LIN {X 0,Y 474.954,Z 430.095,A -85,B 0,C 180,E1 -7279.666,E2 -7279.666} C_VEL
LIN {X 0,Y 474.759,Z 438.387,A -85,B 0,C 180,E1 -7280.308,E2 -7280.308} C_VEL
LIN {X 0,Y 474.498,Z 446.259,A -85,B 0,C 180,E1 -7281.055,E2 -7281.055} C_VEL
LIN {X 0,Y 474.238,Z 453.634,A -85,B 0,C 180,E1 -7281.908,E2 -7281.908} C_VEL
LIN {X 0,Y 474.053,Z 461.103,A -85,B 0,C 180,E1 -7282.976,E2 -7282.976} C_VEL
LIN {X 0,Y 473.911,Z 466.922,A -85,B 0,C 180,E1 -7284.043,E2 -7284.043} C_VEL
LIN {X 0,Y 473.866,Z 470.746,A -85,B 0,C 180,E1 -7284.896,E2 -7284.896} C_VEL
LIN {X 0,Y 473.815,Z 475.078,A -85,B 0,C 180,E1 -7286.174,E2 -7286.174} C_VEL
LIN {X 0,Y 473.748,Z 478.099,A -85,B 0,C 180,E1 -7287.451,E2 -7287.451} C_VEL
LIN {X 0,Y 473.726,Z 479.418,A -85,B 0,C 180,E1 -7288.301,E2 -7288.301} C_VEL
LIN {X 0,Y 473.69,Z 480.236,A -85,B 0,C 180,E1 -7289.151,E2 -7289.151} C_VEL
LIN {X 0,Y 473.674,Z 480.528,A -85,B 0,C 180,E1 -7290.001,E2 -7290.001} C_VEL
LIN {X 0,Y 473.69,Z 480.211,A -85,B 0,C 180,E1 -7290.852,E2 -7290.852} C_VEL
LIN {X 0,Y 473.726,Z 479.389,A -85,B 0,C 180,E1 -7291.702,E2 -7291.702} C_VEL
LIN {X 0,Y 473.748,Z 478.065,A -85,B 0,C 180,E1 -7292.552,E2 -7292.552} C_VEL
LIN {X 0,Y 473.799,Z 475.012,A -85,B 0,C 180,E1 -7293.829,E2 -7293.829} C_VEL
LIN {X 0,Y 473.792,Z 472.221,A -85,B 0,C 180,E1 -7294.681,E2 -7294.681} C_VEL
LIN {X 0,Y 473.911,Z 468.787,A -85,B 0,C 180,E1 -7295.533,E2 -7295.533} C_VEL
LIN {X 0,Y 473.95,Z 463.866,A -85,B 0,C 180,E1 -7296.52,E2 -7296.52} C_VEL
LIN {X 0,Y 474.145,Z 458.151,A -85,B 0,C 180,E1 -7297.453,E2 -7297.453} C_VEL
LIN {X 0,Y 474.275,Z 451.812,A -85,B 0,C 180,E1 -7298.308,E2 -7298.308} C_VEL
LIN {X 0,Y 474.514,Z 444.11,A -85,B 0,C 180,E1 -7299.163,E2 -7299.163} C_VEL
LIN {X 0,Y 474.846,Z 434.562,A -85,B 0,C 180,E1 -7300.016,E2 -7300.016} C_VEL
LIN {X 0,Y 475.091,Z 425.305,A -85,B 0,C 180,E1 -7300.657,E2 -7300.657} C_VEL
LIN {X 0,Y 475.426,Z 415.239,A -85,B 0,C 180,E1 -7301.189,E2 -7301.189} C_VEL
LIN {X 0,Y 475.61,Z 405.755,A -85,B 0,C 180,E1 -7301.562,E2 -7301.562} C_VEL
LIN {X 0,Y 475.842,Z 395.844,A -85,B 0,C 180,E1 -7301.827,E2 -7301.827} C_VEL
LIN {X 0,Y 476.275,Z 333.715,A -85,B 0,C 180,E1 -7302.911,E2 -7302.911} C_VEL
LIN {X 0,Y 474.456,Z 318.892,A -85,B 0,C 180,E1 -7303.244,E2 -7303.244} C_VEL
LIN {X 0,Y 474.728,Z 301.496,A -85,B 0,C 180,E1 -7306.338,E2 -7306.338} C_VEL
LIN {X 0,Y 475.004,Z 283.808,A -85,B 0,C 180,E1 -7309.446,E2 -7309.446} C_VEL
LIN {X 0,Y 475.142,Z 269.646,A -85,B 0,C 180,E1 -7311.932,E2 -7311.932} C_VEL
LIN {X 0,Y 474.695,Z 266.173,A -85,B 0,C 180,E1 -7312.584,E2 -7312.584} C_VEL
LIN {X 0,Y 474.603,Z 266.18,A -85,B 0,C 180,E1 -7315.433,E2 -7315.433} C_VEL
LIN {X 0,Y 474.599,Z 266.182,A -85,B 0,C 180,E1 -7318.287,E2 -7318.287} C_VEL
LIN {X 0,Y 474.581,Z 266.183,A -85,B 0,C 180,E1 -7321.22,E2 -7321.22} C_VEL
LIN {X 0,Y 474.56,Z 266.183,A -85,B 0,C 180,E1 -7324.248,E2 -7324.248} C_VEL
LIN {X 0,Y 474.541,Z 266.185,A -85,B 0,C 180,E1 -7327.39,E2 -7327.39} C_VEL
LIN {X 0,Y 474.591,Z 266.176,A -85,B 0,C 180,E1 -7329.639,E2 -7329.639} C_VEL
LIN {X 0,Y 474.579,Z 266.185,A -85,B 0,C 180,E1 -7332.939,E2 -7332.939} C_VEL
LIN {X 0,Y 474.581,Z 266.177,A -85,B 0,C 180,E1 -7335.889,E2 -7335.889} C_VEL
LIN {X 0,Y 474.614,Z 266.179,A -85,B 0,C 180,E1 -7339.044,E2 -7339.044} C_VEL
LIN {X 0,Y 474.609,Z 266.173,A -85,B 0,C 180,E1 -7341.706,E2 -7341.706} C_VEL
LIN {X 0,Y 474.632,Z 266.174,A -85,B 0,C 180,E1 -7344.723,E2 -7344.723} C_VEL
LIN {X 0,Y 474.642,Z 266.172,A -85,B 0,C 180,E1 -7347.785,E2 -7347.785} C_VEL
LIN {X 0,Y 474.616,Z 266.179,A -85,B 0,C 180,E1 -7350.888,E2 -7350.888} C_VEL
LIN {X 0,Y 474.618,Z 266.179,A -85,B 0,C 180,E1 -7353.623,E2 -7353.623} C_VEL
LIN {X 0,Y 474.649,Z 266.175,A -85,B 0,C 180,E1 -7356.64,E2 -7356.64} C_VEL
LIN {X 0,Y 474.668,Z 266.169,A -85,B 0,C 180,E1 -7360.087,E2 -7360.087} C_VEL
LIN {X 0,Y 474.765,Z 266.163,A -85,B 0,C 180,E1 -7363.661,E2 -7363.661} C_VEL
LIN {X 0,Y 474.843,Z 266.317,A -85,B 0,C 180,E1 -7364.133,E2 -7364.133} C_VEL
LIN {X 0,Y 474.62,Z 284.701,A -85,B 0,C 180,E1 -7366.779,E2 -7366.779} C_VEL
LIN {X 0,Y 476.599,Z 298.432,A -85,B 0,C 180,E1 -7367.103,E2 -7367.103} C_VEL
LIN {X 0,Y 475.902,Z 364.749,A -85,B 0,C 180,E1 -7368.281,E2 -7368.281} C_VEL
LIN {X 0,Y 475.7,Z 376.754,A -85,B 0,C 180,E1 -7368.653,E2 -7368.653} C_VEL
LIN {X 0,Y 475.451,Z 386.848,A -85,B 0,C 180,E1 -7369.133,E2 -7369.133} C_VEL
LIN {X 0,Y 475.243,Z 395.471,A -85,B 0,C 180,E1 -7369.667,E2 -7369.667} C_VEL
LIN {X 0,Y 475.08,Z 403.741,A -85,B 0,C 180,E1 -7370.309,E2 -7370.309} C_VEL
LIN {X 0,Y 474.834,Z 411.591,A -85,B 0,C 180,E1 -7371.056,E2 -7371.056} C_VEL
LIN {X 0,Y 474.563,Z 418.93,A -85,B 0,C 180,E1 -7371.908,E2 -7371.908} C_VEL
LIN {X 0,Y 474.314,Z 427.087,A -85,B 0,C 180,E1 -7373.102,E2 -7373.102} C_VEL
LIN {X 0,Y 474.192,Z 432.129,A -85,B 0,C 180,E1 -7374.041,E2 -7374.041} C_VEL
LIN {X 0,Y 473.929,Z 435.928,A -85,B 0,C 180,E1 -7374.891,E2 -7374.891} C_VEL
LIN {X 0,Y 474.022,Z 438.984,A -85,B 0,C 180,E1 -7375.745,E2 -7375.745} C_VEL
LIN {X 0,Y 473.909,Z 441.375,A -85,B 0,C 180,E1 -7376.595,E2 -7376.595} C_VEL
LIN {X 0,Y 473.83,Z 443.205,A -85,B 0,C 180,E1 -7377.446,E2 -7377.446} C_VEL
LIN {X 0,Y 473.763,Z 444.517,A -85,B 0,C 180,E1 -7378.296,E2 -7378.296} C_VEL
LIN {X 0,Y 473.693,Z 445.334,A -85,B 0,C 180,E1 -7379.146,E2 -7379.146} C_VEL
LIN {X 0,Y 473.676,Z 445.624,A -85,B 0,C 180,E1 -7379.996,E2 -7379.996} C_VEL
LIN {X 0,Y 473.693,Z 445.313,A -85,B 0,C 180,E1 -7380.846,E2 -7380.846} C_VEL
LIN {X 0,Y 473.76,Z 444.504,A -85,B 0,C 180,E1 -7381.696,E2 -7381.696} C_VEL
LIN {X 0,Y 473.804,Z 443.201,A -85,B 0,C 180,E1 -7382.546,E2 -7382.546} C_VEL
LIN {X 0,Y 473.934,Z 440.192,A -85,B 0,C 180,E1 -7383.822,E2 -7383.822} C_VEL
LIN {X 0,Y 473.923,Z 437.448,A -85,B 0,C 180,E1 -7384.674,E2 -7384.674} C_VEL
LIN {X 0,Y 474.009,Z 434.063,A -85,B 0,C 180,E1 -7385.526,E2 -7385.526} C_VEL
LIN {X 0,Y 474.304,Z 429.112,A -85,B 0,C 180,E1 -7386.525,E2 -7386.525} C_VEL
LIN {X 0,Y 474.322,Z 423.544,A -85,B 0,C 180,E1 -7387.444,E2 -7387.444} C_VEL
LIN {X 0,Y 474.513,Z 417.257,A -85,B 0,C 180,E1 -7388.298,E2 -7388.298} C_VEL
LIN {X 0,Y 474.764,Z 410.645,A -85,B 0,C 180,E1 -7389.044,E2 -7389.044} C_VEL
LIN {X 0,Y 475.018,Z 402.647,A -85,B 0,C 180,E1 -7389.791,E2 -7389.791} C_VEL
LIN {X 0,Y 475.318,Z 392.671,A -85,B 0,C 180,E1 -7390.538,E2 -7390.538} C_VEL
LIN {X 0,Y 475.531,Z 382.089,A -85,B 0,C 180,E1 -7391.126,E2 -7391.126} C_VEL
LIN {X 0,Y 475.702,Z 372.217,A -85,B 0,C 180,E1 -7391.527,E2 -7391.527} C_VEL
LIN {X 0,Y 475.842,Z 362.639,A -85,B 0,C 180,E1 -7391.793,E2 -7391.793} C_VEL
LIN {X 0,Y 476.251,Z 297.517,A -85,B 0,C 180,E1 -7392.905,E2 -7392.905} C_VEL
LIN {X 0,Y 474.524,Z 286.851,A -85,B 0,C 180,E1 -7393.15,E2 -7393.15} C_VEL
LIN {X 0,Y 474.786,Z 274.007,A -85,B 0,C 180,E1 -7396.329,E2 -7396.329} C_VEL
LIN {X 0,Y 474.746,Z 266.283,A -85,B 0,C 180,E1 -7398.3,E2 -7398.3} C_VEL
LIN {X 0,Y 474.623,Z 266.177,A -85,B 0,C 180,E1 -7401.111,E2 -7401.111} C_VEL
LIN {X 0,Y 474.61,Z 266.177,A -85,B 0,C 180,E1 -7404.489,E2 -7404.489} C_VEL
LIN {X 0,Y 474.582,Z 266.182,A -85,B 0,C 180,E1 -7407.321,E2 -7407.321} C_VEL
LIN {X 0,Y 474.574,Z 266.18,A -85,B 0,C 180,E1 -7410.226,E2 -7410.226} C_VEL
LIN {X 0,Y 474.611,Z 266.179,A -85,B 0,C 180,E1 -7413.215,E2 -7413.215} C_VEL
LIN {X 0,Y 474.557,Z 266.182,A -85,B 0,C 180,E1 -7416.319,E2 -7416.319} C_VEL
LIN {X 0,Y 474.595,Z 266.181,A -85,B 0,C 180,E1 -7419.543,E2 -7419.543} C_VEL
LIN {X 0,Y 474.568,Z 266.182,A -85,B 0,C 180,E1 -7422.228,E2 -7422.228} C_VEL
LIN {X 0,Y 474.582,Z 266.183,A -85,B 0,C 180,E1 -7425.293,E2 -7425.293} C_VEL
LIN {X 0,Y 474.584,Z 266.182,A -85,B 0,C 180,E1 -7428.209,E2 -7428.209} C_VEL
LIN {X 0,Y 474.571,Z 266.185,A -85,B 0,C 180,E1 -7431.538,E2 -7431.538} C_VEL
LIN {X 0,Y 474.586,Z 266.179,A -85,B 0,C 180,E1 -7434.721,E2 -7434.721} C_VEL
LIN {X 0,Y 474.591,Z 266.182,A -85,B 0,C 180,E1 -7437.783,E2 -7437.783} C_VEL
LIN {X 0,Y 474.553,Z 266.183,A -85,B 0,C 180,E1 -7438.959,E2 -7438.959} C_VEL
LIN {X 0,Y 473.909,Z 266.266,A -85,B 0,C 180,E1 -7439.668,E2 -7439.668} C_VEL
LIN {X 0,Y 471.103,Z 266.616,A -85,B 0,C 180,E1 -7440.819,E2 -7440.819} C_VEL
LIN {X 0,Y 468.712,Z 266.915,A -85,B 0,C 180,E1 -7441.747,E2 -7441.747} C_VEL
LIN {X 0,Y 467.671,Z 267.043,A -85,B 0,C 180,E1 -7442.463,E2 -7442.463} C_VEL
LIN {X 0,Y 467.58,Z 267.053,A -85,B 0,C 180,E1 -7442.706,E2 -7442.706} C_VEL
LIN {X 0,Y 467.554,Z 267.055,A -85,B 0,C 180,E1 -7445.109,E2 -7445.109} C_VEL
LIN {X 0,Y 467.482,Z 267.067,A -85,B 0,C 180,E1 -7447.922,E2 -7447.922} C_VEL
LIN {X 0,Y 467.569,Z 267.056,A -85,B 0,C 180,E1 -7450.689,E2 -7450.689} C_VEL
LIN {X 0,Y 467.594,Z 267.054,A -85,B 0,C 180,E1 -7454.112,E2 -7454.112} C_VEL
LIN {X 0,Y 467.641,Z 267.045,A -85,B 0,C 180,E1 -7457.853,E2 -7457.853} C_VEL
LIN {X 0,Y 467.626,Z 267.047,A -85,B 0,C 180,E1 -7461.355,E2 -7461.355} C_VEL
LIN {X 0,Y 467.694,Z 267.038,A -85,B 0,C 180,E1 -7463.961,E2 -7463.961} C_VEL
LIN {X 0,Y 467.808,Z 267.025,A -85,B 0,C 180,E1 -7467.415,E2 -7467.415} C_VEL
LIN {X 0,Y 467.82,Z 267.022,A -85,B 0,C 180,E1 -7469.999,E2 -7469.999} C_VEL
LIN {X 0,Y 467.807,Z 267.027,A -85,B 0,C 180,E1 -7472.582,E2 -7472.582} C_VEL
LIN {X 0,Y 467.692,Z 267.038,A -85,B 0,C 180,E1 -7476.036,E2 -7476.036} C_VEL
LIN {X 0,Y 467.628,Z 267.048,A -85,B 0,C 180,E1 -7478.642,E2 -7478.642} C_VEL
LIN {X 0,Y 467.637,Z 267.044,A -85,B 0,C 180,E1 -7482.144,E2 -7482.144} C_VEL
LIN {X 0,Y 467.587,Z 267.052,A -85,B 0,C 180,E1 -7485.885,E2 -7485.885} C_VEL
LIN {X 0,Y 467.563,Z 267.057,A -85,B 0,C 180,E1 -7489.309,E2 -7489.309} C_VEL
LIN {X 0,Y 467.479,Z 267.066,A -85,B 0,C 180,E1 -7492.075,E2 -7492.075} C_VEL
LIN {X 0,Y 467.554,Z 267.056,A -85,B 0,C 180,E1 -7494.888,E2 -7494.888} C_VEL
LIN {X 0,Y 467.57,Z 267.055,A -85,B 0,C 180,E1 -7497.77,E2 -7497.77} C_VEL
LIN {X 0,Y 467.515,Z 267.061,A -85,B 0,C 180,E1 -7501.048,E2 -7501.048} C_VEL
LIN {X 0,Y 467.534,Z 267.06,A -85,B 0,C 180,E1 -7504.245,E2 -7504.245} C_VEL
LIN {X 0,Y 467.497,Z 267.063,A -85,B 0,C 180,E1 -7507.19,E2 -7507.19} C_VEL
LIN {X 0,Y 467.55,Z 267.058,A -85,B 0,C 180,E1 -7510.265,E2 -7510.265} C_VEL
LIN {X 0,Y 467.568,Z 267.055,A -85,B 0,C 180,E1 -7512.574,E2 -7512.574} C_VEL
LIN {X 0,Y 467.525,Z 267.061,A -85,B 0,C 180,E1 -7516.18,E2 -7516.18} C_VEL
LIN {X 0,Y 467.542,Z 267.058,A -85,B 0,C 180,E1 -7518.725,E2 -7518.725} C_VEL
LIN {X 0,Y 467.528,Z 267.058,A -85,B 0,C 180,E1 -7521.411,E2 -7521.411} C_VEL
LIN {X 0,Y 467.52,Z 267.062,A -85,B 0,C 180,E1 -7524.264,E2 -7524.264} C_VEL
LIN {X 0,Y 467.541,Z 267.056,A -85,B 0,C 180,E1 -7527.325,E2 -7527.325} C_VEL
LIN {X 0,Y 467.529,Z 267.06,A -85,B 0,C 180,E1 -7530.672,E2 -7530.672} C_VEL
LIN {X 0,Y 467.55,Z 267.057,A -85,B 0,C 180,E1 -7533.202,E2 -7533.202} C_VEL
LIN {X 0,Y 467.555,Z 267.059,A -85,B 0,C 180,E1 -7536.474,E2 -7536.474} C_VEL
LIN {X 0,Y 467.589,Z 267.05,A -85,B 0,C 180,E1 -7539.781,E2 -7539.781} C_VEL
LIN {X 0,Y 467.566,Z 267.057,A -85,B 0,C 180,E1 -7542.511,E2 -7542.511} C_VEL
LIN {X 0,Y 467.575,Z 267.055,A -85,B 0,C 180,E1 -7545.201,E2 -7545.201} C_VEL
LIN {X 0,Y 467.629,Z 267.045,A -85,B 0,C 180,E1 -7547.859,E2 -7547.859} C_VEL
LIN {X 0,Y 467.644,Z 267.046,A -85,B 0,C 180,E1 -7551.361,E2 -7551.361} C_VEL
LIN {X 0,Y 467.704,Z 267.036,A -85,B 0,C 180,E1 -7553.967,E2 -7553.967} C_VEL
LIN {X 0,Y 467.801,Z 267.027,A -85,B 0,C 180,E1 -7557.421,E2 -7557.421} C_VEL
LIN {X 0,Y 467.831,Z 267.021,A -85,B 0,C 180,E1 -7560.004,E2 -7560.004} C_VEL
LIN {X 0,Y 467.831,Z 267.02,A -85,B 0,C 180,E1 -7562.587,E2 -7562.587} C_VEL
LIN {X 0,Y 467.696,Z 267.039,A -85,B 0,C 180,E1 -7566.042,E2 -7566.042} C_VEL
LIN {X 0,Y 467.653,Z 267.042,A -85,B 0,C 180,E1 -7568.647,E2 -7568.647} C_VEL
LIN {X 0,Y 467.644,Z 267.046,A -85,B 0,C 180,E1 -7572.149,E2 -7572.149} C_VEL
LIN {X 0,Y 467.602,Z 267.052,A -85,B 0,C 180,E1 -7575.7,E2 -7575.7} C_VEL
LIN {X 0,Y 467.61,Z 267.05,A -85,B 0,C 180,E1 -7579.312,E2 -7579.312} C_VEL
LIN {X 0,Y 467.523,Z 267.061,A -85,B 0,C 180,E1 -7582.078,E2 -7582.078} C_VEL
LIN {X 0,Y 467.552,Z 267.055,A -85,B 0,C 180,E1 -7584.893,E2 -7584.893} C_VEL
LIN {X 0,Y 467.573,Z 267.057,A -85,B 0,C 180,E1 -7587.775,E2 -7587.775} C_VEL
LIN {X 0,Y 467.562,Z 267.054,A -85,B 0,C 180,E1 -7591.048,E2 -7591.048} C_VEL
LIN {X 0,Y 467.571,Z 267.056,A -85,B 0,C 180,E1 -7594.243,E2 -7594.243} C_VEL
LIN {X 0,Y 467.518,Z 267.059,A -85,B 0,C 180,E1 -7597.185,E2 -7597.185} C_VEL
LIN {X 0,Y 467.553,Z 267.059,A -85,B 0,C 180,E1 -7600.27,E2 -7600.27} C_VEL
LIN {X 0,Y 467.544,Z 267.056,A -85,B 0,C 180,E1 -7603.749,E2 -7603.749} C_VEL
LIN {X 0,Y 467.531,Z 267.062,A -85,B 0,C 180,E1 -7606.256,E2 -7606.256} C_VEL
LIN {X 0,Y 467.556,Z 267.054,A -85,B 0,C 180,E1 -7609.736,E2 -7609.736} C_VEL
LIN {X 0,Y 467.537,Z 267.06,A -85,B 0,C 180,E1 -7612.818,E2 -7612.818} C_VEL
LIN {X 0,Y 467.576,Z 267.052,A -85,B 0,C 180,E1 -7615.763,E2 -7615.763} C_VEL
LIN {X 0,Y 467.543,Z 267.059,A -85,B 0,C 180,E1 -7618.963,E2 -7618.963} C_VEL
LIN {X 0,Y 467.545,Z 267.056,A -85,B 0,C 180,E1 -7622.228,E2 -7622.228} C_VEL
LIN {X 0,Y 467.59,Z 267.057,A -85,B 0,C 180,E1 -7625.588,E2 -7625.588} C_VEL
LIN {X 0,Y 467.624,Z 267.185,A -85,B 0,C 180,E1 -7625.885,E2 -7625.885} C_VEL
LIN {X 0,Y 468.989,Z 275.944,A -85,B 0,C 180,E1 -7627.768,E2 -7627.768} C_VEL
LIN {X 0,Y 468.477,Z 290.486,A -85,B 0,C 180,E1 -7630.731,E2 -7630.731} C_VEL
LIN {X 0,Y 467.831,Z 306.981,A -85,B 0,C 180,E1 -7634.042,E2 -7634.042} C_VEL
LIN {X 0,Y 467.465,Z 320.443,A -85,B 0,C 180,E1 -7636.695,E2 -7636.695} C_VEL
LIN {X 0,Y 469.327,Z 337.479,A -85,B 0,C 180,E1 -7637.043,E2 -7637.043} C_VEL
LIN {X 0,Y 468.775,Z 398.013,A -85,B 0,C 180,E1 -7638.105,E2 -7638.105} C_VEL
LIN {X 0,Y 468.531,Z 408.917,A -85,B 0,C 180,E1 -7638.428,E2 -7638.428} C_VEL
LIN {X 0,Y 468.221,Z 420.685,A -85,B 0,C 180,E1 -7638.968,E2 -7638.968} C_VEL
LIN {X 0,Y 467.929,Z 429.416,A -85,B 0,C 180,E1 -7639.509,E2 -7639.509} C_VEL
LIN {X 0,Y 467.709,Z 437.792,A -85,B 0,C 180,E1 -7640.16,E2 -7640.16} C_VEL
LIN {X 0,Y 467.41,Z 445.729,A -85,B 0,C 180,E1 -7640.918,E2 -7640.918} C_VEL
LIN {X 0,Y 467.18,Z 453.162,A -85,B 0,C 180,E1 -7641.785,E2 -7641.785} C_VEL
LIN {X 0,Y 466.996,Z 460.696,A -85,B 0,C 180,E1 -7642.869,E2 -7642.869} C_VEL
LIN {X 0,Y 466.822,Z 466.563,A -85,B 0,C 180,E1 -7643.952,E2 -7643.952} C_VEL
LIN {X 0,Y 466.799,Z 470.41,A -85,B 0,C 180,E1 -7644.819,E2 -7644.819} C_VEL
LIN {X 0,Y 466.706,Z 474.77,A -85,B 0,C 180,E1 -7646.116,E2 -7646.116} C_VEL
LIN {X 0,Y 466.669,Z 477.808,A -85,B 0,C 180,E1 -7647.412,E2 -7647.412} C_VEL
LIN {X 0,Y 466.634,Z 479.14,A -85,B 0,C 180,E1 -7648.275,E2 -7648.275} C_VEL
LIN {X 0,Y 466.621,Z 479.97,A -85,B 0,C 180,E1 -7649.138,E2 -7649.138} C_VEL
LIN {X 0,Y 466.603,Z 480.263,A -85,B 0,C 180,E1 -7650.001,E2 -7650.001} C_VEL
LIN {X 0,Y 466.621,Z 479.951,A -85,B 0,C 180,E1 -7650.864,E2 -7650.864} C_VEL
LIN {X 0,Y 466.634,Z 479.134,A -85,B 0,C 180,E1 -7651.728,E2 -7651.728} C_VEL
LIN {X 0,Y 466.67,Z 477.814,A -85,B 0,C 180,E1 -7652.591,E2 -7652.591} C_VEL
LIN {X 0,Y 466.692,Z 474.769,A -85,B 0,C 180,E1 -7653.887,E2 -7653.887} C_VEL
LIN {X 0,Y 466.72,Z 471.986,A -85,B 0,C 180,E1 -7654.752,E2 -7654.752} C_VEL
LIN {X 0,Y 466.828,Z 468.557,A -85,B 0,C 180,E1 -7655.617,E2 -7655.617} C_VEL
LIN {X 0,Y 466.918,Z 463.079,A -85,B 0,C 180,E1 -7656.719,E2 -7656.719} C_VEL
LIN {X 0,Y 467.092,Z 456.451,A -85,B 0,C 180,E1 -7657.784,E2 -7657.784} C_VEL
LIN {X 0,Y 467.392,Z 448.009,A -85,B 0,C 180,E1 -7658.867,E2 -7658.867} C_VEL
LIN {X 0,Y 467.731,Z 439.338,A -85,B 0,C 180,E1 -7659.733,E2 -7659.733} C_VEL
LIN {X 0,Y 467.913,Z 431.356,A -85,B 0,C 180,E1 -7660.385,E2 -7660.385} C_VEL
LIN {X 0,Y 468.171,Z 423.182,A -85,B 0,C 180,E1 -7660.926,E2 -7660.926} C_VEL
LIN {X 0,Y 468.476,Z 413.81,A -85,B 0,C 180,E1 -7661.412,E2 -7661.412} C_VEL
LIN {X 0,Y 468.683,Z 404.762,A -85,B 0,C 180,E1 -7661.763,E2 -7661.763} C_VEL
LIN {X 0,Y 468.943,Z 394.573,A -85,B 0,C 180,E1 -7662.031,E2 -7662.031} C_VEL
LIN {X 0,Y 469.412,Z 334.466,A -85,B 0,C 180,E1 -7663.116,E2 -7663.116} C_VEL
LIN {X 0,Y 467.446,Z 318.359,A -85,B 0,C 180,E1 -7663.505,E2 -7663.505} C_VEL
LIN {X 0,Y 467.802,Z 298.693,A -85,B 0,C 180,E1 -7667.036,E2 -7667.036} C_VEL
LIN {X 0,Y 468.103,Z 279.668,A -85,B 0,C 180,E1 -7670.432,E2 -7670.432} C_VEL
LIN {X 0,Y 468.156,Z 270.594,A -85,B 0,C 180,E1 -7672.044,E2 -7672.044} C_VEL
LIN {X 0,Y 467.634,Z 267.052,A -85,B 0,C 180,E1 -7672.71,E2 -7672.71} C_VEL
LIN {X 0,Y 467.544,Z 267.058,A -85,B 0,C 180,E1 -7675.845,E2 -7675.845} C_VEL
LIN {X 0,Y 467.535,Z 267.065,A -85,B 0,C 180,E1 -7678.754,E2 -7678.754} C_VEL
LIN {X 0,Y 467.548,Z 267.055,A -85,B 0,C 180,E1 -7681.744,E2 -7681.744} C_VEL
LIN {X 0,Y 467.5,Z 267.066,A -85,B 0,C 180,E1 -7684.839,E2 -7684.839} C_VEL
LIN {X 0,Y 467.546,Z 267.054,A -85,B 0,C 180,E1 -7688.048,E2 -7688.048} C_VEL
LIN {X 0,Y 467.563,Z 267.054,A -85,B 0,C 180,E1 -7691.406,E2 -7691.406} C_VEL
LIN {X 0,Y 467.56,Z 267.058,A -85,B 0,C 180,E1 -7695.049,E2 -7695.049} C_VEL
LIN {X 0,Y 467.575,Z 267.053,A -85,B 0,C 180,E1 -7698.725,E2 -7698.725} C_VEL
LIN {X 0,Y 467.566,Z 267.049,A -85,B 0,C 180,E1 -7701.953,E2 -7701.953} C_VEL
LIN {X 0,Y 467.57,Z 267.056,A -85,B 0,C 180,E1 -7705.165,E2 -7705.165} C_VEL
LIN {X 0,Y 467.593,Z 267.05,A -85,B 0,C 180,E1 -7708.258,E2 -7708.258} C_VEL
LIN {X 0,Y 467.564,Z 267.06,A -85,B 0,C 180,E1 -7711.246,E2 -7711.246} C_VEL
LIN {X 0,Y 467.607,Z 267.051,A -85,B 0,C 180,E1 -7714.395,E2 -7714.395} C_VEL
LIN {X 0,Y 467.591,Z 267.058,A -85,B 0,C 180,E1 -7716.993,E2 -7716.993} C_VEL
LIN {X 0,Y 467.637,Z 267.047,A -85,B 0,C 180,E1 -7719.774,E2 -7719.774} C_VEL
LIN {X 0,Y 467.663,Z 267.045,A -85,B 0,C 180,E1 -7722.505,E2 -7722.505} C_VEL
LIN {X 0,Y 467.769,Z 267.09,A -85,B 0,C 180,E1 -7723.961,E2 -7723.961} C_VEL
LIN {X 0,Y 467.867,Z 271.123,A -85,B 0,C 180,E1 -7724.533,E2 -7724.533} C_VEL
LIN {X 0,Y 467.683,Z 284.995,A -85,B 0,C 180,E1 -7726.543,E2 -7726.543} C_VEL
LIN {X 0,Y 469.763,Z 299.131,A -85,B 0,C 180,E1 -7726.883,E2 -7726.883} C_VEL
LIN {X 0,Y 468.979,Z 365.544,A -85,B 0,C 180,E1 -7728.105,E2 -7728.105} C_VEL
LIN {X 0,Y 468.759,Z 377.239,A -85,B 0,C 180,E1 -7728.483,E2 -7728.483} C_VEL
LIN {X 0,Y 468.501,Z 387.235,A -85,B 0,C 180,E1 -7728.97,E2 -7728.97} C_VEL
LIN {X 0,Y 468.277,Z 395.806,A -85,B 0,C 180,E1 -7729.511,E2 -7729.511} C_VEL
LIN {X 0,Y 468.103,Z 404.073,A -85,B 0,C 180,E1 -7730.163,E2 -7730.163} C_VEL
LIN {X 0,Y 467.834,Z 411.923,A -85,B 0,C 180,E1 -7730.921,E2 -7730.921} C_VEL
LIN {X 0,Y 467.564,Z 419.262,A -85,B 0,C 180,E1 -7731.786,E2 -7731.786} C_VEL
LIN {X 0,Y 467.279,Z 426.809,A -85,B 0,C 180,E1 -7732.89,E2 -7732.89} C_VEL
LIN {X 0,Y 467.161,Z 432.452,A -85,B 0,C 180,E1 -7733.951,E2 -7733.951} C_VEL
LIN {X 0,Y 466.869,Z 436.25,A -85,B 0,C 180,E1 -7734.814,E2 -7734.814} C_VEL
LIN {X 0,Y 466.966,Z 439.307,A -85,B 0,C 180,E1 -7735.68,E2 -7735.68} C_VEL
LIN {X 0,Y 466.843,Z 441.693,A -85,B 0,C 180,E1 -7736.544,E2 -7736.544} C_VEL
LIN {X 0,Y 466.747,Z 443.512,A -85,B 0,C 180,E1 -7737.407,E2 -7737.407} C_VEL
LIN {X 0,Y 466.699,Z 444.81,A -85,B 0,C 180,E1 -7738.27,E2 -7738.27} C_VEL
LIN {X 0,Y 466.624,Z 445.612,A -85,B 0,C 180,E1 -7739.133,E2 -7739.133} C_VEL
LIN {X 0,Y 466.605,Z 445.894,A -85,B 0,C 180,E1 -7739.996,E2 -7739.996} C_VEL
LIN {X 0,Y 466.624,Z 445.57,A -85,B 0,C 180,E1 -7740.859,E2 -7740.859} C_VEL
LIN {X 0,Y 466.667,Z 444.74,A -85,B 0,C 180,E1 -7741.722,E2 -7741.722} C_VEL
LIN {X 0,Y 466.723,Z 443.41,A -85,B 0,C 180,E1 -7742.585,E2 -7742.585} C_VEL
LIN {X 0,Y 466.866,Z 440.372,A -85,B 0,C 180,E1 -7743.88,E2 -7743.88} C_VEL
LIN {X 0,Y 466.845,Z 436.03,A -85,B 0,C 180,E1 -7745.178,E2 -7745.178} C_VEL
LIN {X 0,Y 467.198,Z 430.741,A -85,B 0,C 180,E1 -7746.341,E2 -7746.341} C_VEL
LIN {X 0,Y 467.247,Z 424.998,A -85,B 0,C 180,E1 -7747.341,E2 -7747.341} C_VEL
LIN {X 0,Y 467.439,Z 418.938,A -85,B 0,C 180,E1 -7748.207,E2 -7748.207} C_VEL
LIN {X 0,Y 467.688,Z 411.56,A -85,B 0,C 180,E1 -7749.073,E2 -7749.073} C_VEL
LIN {X 0,Y 467.948,Z 403.683,A -85,B 0,C 180,E1 -7749.832,E2 -7749.832} C_VEL
LIN {X 0,Y 468.18,Z 395.387,A -85,B 0,C 180,E1 -7750.482,E2 -7750.482} C_VEL
LIN {X 0,Y 468.462,Z 384.869,A -85,B 0,C 180,E1 -7751.132,E2 -7751.132} C_VEL
LIN {X 0,Y 468.727,Z 373.722,A -85,B 0,C 180,E1 -7751.618,E2 -7751.618} C_VEL
LIN {X 0,Y 468.864,Z 363.61,A -85,B 0,C 180,E1 -7751.916,E2 -7751.916} C_VEL
LIN {X 0,Y 469.313,Z 298.256,A -85,B 0,C 180,E1 -7753.071,E2 -7753.071} C_VEL
LIN {X 0,Y 467.523,Z 287.081,A -85,B 0,C 180,E1 -7753.325,E2 -7753.325} C_VEL
LIN {X 0,Y 467.793,Z 274.082,A -85,B 0,C 180,E1 -7756.58,E2 -7756.58} C_VEL
LIN {X 0,Y 467.664,Z 267.046,A -85,B 0,C 180,E1 -7758.422,E2 -7758.422} C_VEL
LIN {X 0,Y 467.568,Z 267.056,A -85,B 0,C 180,E1 -7761.262,E2 -7761.262} C_VEL
LIN {X 0,Y 467.54,Z 267.057,A -85,B 0,C 180,E1 -7763.939,E2 -7763.939} C_VEL
LIN {X 0,Y 467.518,Z 267.063,A -85,B 0,C 180,E1 -7766.8,E2 -7766.8} C_VEL
LIN {X 0,Y 467.521,Z 267.061,A -85,B 0,C 180,E1 -7769.734,E2 -7769.734} C_VEL
LIN {X 0,Y 467.559,Z 267.056,A -85,B 0,C 180,E1 -7772.753,E2 -7772.753} C_VEL
LIN {X 0,Y 467.525,Z 267.061,A -85,B 0,C 180,E1 -7775.884,E2 -7775.884} C_VEL
LIN {X 0,Y 467.525,Z 267.062,A -85,B 0,C 180,E1 -7779.142,E2 -7779.142} C_VEL
LIN {X 0,Y 467.542,Z 267.06,A -85,B 0,C 180,E1 -7781.398,E2 -7781.398} C_VEL
LIN {X 0,Y 467.531,Z 267.059,A -85,B 0,C 180,E1 -7785.047,E2 -7785.047} C_VEL
LIN {X 0,Y 467.554,Z 267.059,A -85,B 0,C 180,E1 -7787.435,E2 -7787.435} C_VEL
LIN {X 0,Y 467.52,Z 267.059,A -85,B 0,C 180,E1 -7790.848,E2 -7790.848} C_VEL
LIN {X 0,Y 467.52,Z 267.062,A -85,B 0,C 180,E1 -7794.256,E2 -7794.256} C_VEL
LIN {X 0,Y 467.538,Z 267.058,A -85,B 0,C 180,E1 -7797.316,E2 -7797.316} C_VEL
LIN {X 0,Y 467.524,Z 267.06,A -85,B 0,C 180,E1 -7800.663,E2 -7800.663} C_VEL
LIN {X 0,Y 467.58,Z 267.053,A -85,B 0,C 180,E1 -7802.706,E2 -7802.706} C_VEL
LIN {X 0,Y 466.886,Z 267.139,A -85,B 0,C 180,E1 -7803.424,E2 -7803.424} C_VEL
LIN {X 0,Y 464,Z 267.501,A -85,B 0,C 180,E1 -7804.591,E2 -7804.591} C_VEL
LIN {X 0,Y 461.583,Z 267.801,A -85,B 0,C 180,E1 -7805.531,E2 -7805.531} C_VEL
LIN {X 0,Y 460.564,Z 267.928,A -85,B 0,C 180,E1 -7806.258,E2 -7806.258} C_VEL
LIN {X 0,Y 460.49,Z 267.937,A -85,B 0,C 180,E1 -7806.504,E2 -7806.504} C_VEL
LIN {X 0,Y 460.498,Z 267.934,A -85,B 0,C 180,E1 -7809.449,E2 -7809.449} C_VEL
LIN {X 0,Y 460.504,Z 267.936,A -85,B 0,C 180,E1 -7812.227,E2 -7812.227} C_VEL
LIN {X 0,Y 460.509,Z 267.935,A -85,B 0,C 180,E1 -7814.962,E2 -7814.962} C_VEL
LIN {X 0,Y 460.602,Z 267.921,A -85,B 0,C 180,E1 -7817.664,E2 -7817.664} C_VEL
LIN {X 0,Y 460.573,Z 267.926,A -85,B 0,C 180,E1 -7821.221,E2 -7821.221} C_VEL
LIN {X 0,Y 460.658,Z 267.914,A -85,B 0,C 180,E1 -7823.868,E2 -7823.868} C_VEL
LIN {X 0,Y 460.774,Z 267.901,A -85,B 0,C 180,E1 -7827.376,E2 -7827.376} C_VEL
LIN {X 0,Y 460.791,Z 267.897,A -85,B 0,C 180,E1 -7829.999,E2 -7829.999} C_VEL
LIN {X 0,Y 460.773,Z 267.904,A -85,B 0,C 180,E1 -7832.621,E2 -7832.621} C_VEL
LIN {X 0,Y 460.656,Z 267.914,A -85,B 0,C 180,E1 -7836.129,E2 -7836.129} C_VEL
LIN {X 0,Y 460.574,Z 267.928,A -85,B 0,C 180,E1 -7838.776,E2 -7838.776} C_VEL
LIN {X 0,Y 460.573,Z 267.925,A -85,B 0,C 180,E1 -7842.457,E2 -7842.457} C_VEL
LIN {X 0,Y 460.539,Z 267.93,A -85,B 0,C 180,E1 -7845.998,E2 -7845.998} C_VEL
LIN {X 0,Y 460.51,Z 267.935,A -85,B 0,C 180,E1 -7848.902,E2 -7848.902} C_VEL
LIN {X 0,Y 460.457,Z 267.941,A -85,B 0,C 180,E1 -7851.487,E2 -7851.487} C_VEL
LIN {X 0,Y 460.488,Z 267.936,A -85,B 0,C 180,E1 -7854.333,E2 -7854.333} C_VEL
LIN {X 0,Y 460.526,Z 267.934,A -85,B 0,C 180,E1 -7857.245,E2 -7857.245} C_VEL
LIN {X 0,Y 460.469,Z 267.939,A -85,B 0,C 180,E1 -7860.241,E2 -7860.241} C_VEL
LIN {X 0,Y 460.473,Z 267.94,A -85,B 0,C 180,E1 -7863.327,E2 -7863.327} C_VEL
LIN {X 0,Y 460.425,Z 267.944,A -85,B 0,C 180,E1 -7866.532,E2 -7866.532} C_VEL
LIN {X 0,Y 460.534,Z 267.932,A -85,B 0,C 180,E1 -7869.86,E2 -7869.86} C_VEL
LIN {X 0,Y 460.491,Z 267.935,A -85,B 0,C 180,E1 -7872.907,E2 -7872.907} C_VEL
LIN {X 0,Y 460.474,Z 267.941,A -85,B 0,C 180,E1 -7875.832,E2 -7875.832} C_VEL
LIN {X 0,Y 460.496,Z 267.935,A -85,B 0,C 180,E1 -7878.994,E2 -7878.994} C_VEL
LIN {X 0,Y 460.498,Z 267.934,A -85,B 0,C 180,E1 -7881.272,E2 -7881.272} C_VEL
LIN {X 0,Y 460.47,Z 267.94,A -85,B 0,C 180,E1 -7884.559,E2 -7884.559} C_VEL
LIN {X 0,Y 460.49,Z 267.935,A -85,B 0,C 180,E1 -7887.72,E2 -7887.72} C_VEL
LIN {X 0,Y 460.499,Z 267.936,A -85,B 0,C 180,E1 -7890.773,E2 -7890.773} C_VEL
LIN {X 0,Y 460.505,Z 267.933,A -85,B 0,C 180,E1 -7893.738,E2 -7893.738} C_VEL
LIN {X 0,Y 460.509,Z 267.935,A -85,B 0,C 180,E1 -7896.628,E2 -7896.628} C_VEL
LIN {X 0,Y 460.518,Z 267.932,A -85,B 0,C 180,E1 -7899.457,E2 -7899.457} C_VEL
LIN {X 0,Y 460.517,Z 267.933,A -85,B 0,C 180,E1 -7902.234,E2 -7902.234} C_VEL
LIN {X 0,Y 460.535,Z 267.932,A -85,B 0,C 180,E1 -7904.969,E2 -7904.969} C_VEL
LIN {X 0,Y 460.583,Z 267.926,A -85,B 0,C 180,E1 -7908.564,E2 -7908.564} C_VEL
LIN {X 0,Y 460.594,Z 267.924,A -85,B 0,C 180,E1 -7911.228,E2 -7911.228} C_VEL
LIN {X 0,Y 460.67,Z 267.913,A -85,B 0,C 180,E1 -7913.874,E2 -7913.874} C_VEL
LIN {X 0,Y 460.745,Z 267.905,A -85,B 0,C 180,E1 -7917.382,E2 -7917.382} C_VEL
LIN {X 0,Y 460.801,Z 267.897,A -85,B 0,C 180,E1 -7920.004,E2 -7920.004} C_VEL
LIN {X 0,Y 460.772,Z 267.9,A -85,B 0,C 180,E1 -7922.627,E2 -7922.627} C_VEL
LIN {X 0,Y 460.661,Z 267.915,A -85,B 0,C 180,E1 -7926.135,E2 -7926.135} C_VEL
LIN {X 0,Y 460.603,Z 267.921,A -85,B 0,C 180,E1 -7928.781,E2 -7928.781} C_VEL
LIN {X 0,Y 460.586,Z 267.923,A -85,B 0,C 180,E1 -7932.439,E2 -7932.439} C_VEL
LIN {X 0,Y 460.547,Z 267.93,A -85,B 0,C 180,E1 -7935.982,E2 -7935.982} C_VEL
LIN {X 0,Y 460.557,Z 267.93,A -85,B 0,C 180,E1 -7939.62,E2 -7939.62} C_VEL
LIN {X 0,Y 460.499,Z 267.936,A -85,B 0,C 180,E1 -7942.433,E2 -7942.433} C_VEL
LIN {X 0,Y 460.528,Z 267.934,A -85,B 0,C 180,E1 -7945.797,E2 -7945.797} C_VEL
LIN {X 0,Y 460.519,Z 267.933,A -85,B 0,C 180,E1 -7948.238,E2 -7948.238} C_VEL
LIN {X 0,Y 460.516,Z 267.932,A -85,B 0,C 180,E1 -7951.286,E2 -7951.286} C_VEL
LIN {X 0,Y 460.516,Z 267.934,A -85,B 0,C 180,E1 -7954.506,E2 -7954.506} C_VEL
LIN {X 0,Y 460.482,Z 267.937,A -85,B 0,C 180,E1 -7957.628,E2 -7957.628} C_VEL
LIN {X 0,Y 460.512,Z 267.933,A -85,B 0,C 180,E1 -7961.016,E2 -7961.016} C_VEL
LIN {X 0,Y 460.509,Z 267.935,A -85,B 0,C 180,E1 -7964.593,E2 -7964.593} C_VEL
LIN {X 0,Y 460.473,Z 267.937,A -85,B 0,C 180,E1 -7967.816,E2 -7967.816} C_VEL
LIN {X 0,Y 460.51,Z 267.934,A -85,B 0,C 180,E1 -7970.138,E2 -7970.138} C_VEL
LIN {X 0,Y 460.47,Z 267.938,A -85,B 0,C 180,E1 -7973.472,E2 -7973.472} C_VEL
LIN {X 0,Y 460.517,Z 267.935,A -85,B 0,C 180,E1 -7976.677,E2 -7976.677} C_VEL
LIN {X 0,Y 460.498,Z 267.934,A -85,B 0,C 180,E1 -7979.761,E2 -7979.761} C_VEL
LIN {X 0,Y 460.49,Z 267.939,A -85,B 0,C 180,E1 -7982.753,E2 -7982.753} C_VEL
LIN {X 0,Y 460.598,Z 268.099,A -85,B 0,C 180,E1 -7985.758,E2 -7985.758} C_VEL
LIN {X 0,Y 461.997,Z 276.748,A -85,B 0,C 180,E1 -7987.649,E2 -7987.649} C_VEL
LIN {X 0,Y 461.477,Z 290.16,A -85,B 0,C 180,E1 -7990.427,E2 -7990.427} C_VEL
LIN {X 0,Y 460.816,Z 307.258,A -85,B 0,C 180,E1 -7993.914,E2 -7993.914} C_VEL
LIN {X 0,Y 460.411,Z 320.129,A -85,B 0,C 180,E1 -7996.513,E2 -7996.513} C_VEL
LIN {X 0,Y 462.374,Z 337.03,A -85,B 0,C 180,E1 -7996.871,E2 -7996.871} C_VEL
LIN {X 0,Y 461.785,Z 398.398,A -85,B 0,C 180,E1 -7997.978,E2 -7997.978} C_VEL
LIN {X 0,Y 461.477,Z 410.482,A -85,B 0,C 180,E1 -7998.36,E2 -7998.36} C_VEL
LIN {X 0,Y 461.156,Z 421.58,A -85,B 0,C 180,E1 -7998.909,E2 -7998.909} C_VEL
LIN {X 0,Y 460.851,Z 430.085,A -85,B 0,C 180,E1 -7999.457,E2 -7999.457} C_VEL
LIN {X 0,Y 460.64,Z 438.3,A -85,B 0,C 180,E1 -8000.118,E2 -8000.118} C_VEL
LIN {X 0,Y 460.325,Z 446.112,A -85,B 0,C 180,E1 -8000.888,E2 -8000.888} C_VEL
LIN {X 0,Y 460.071,Z 454.314,A -85,B 0,C 180,E1 -8001.878,E2 -8001.878} C_VEL
LIN {X 0,Y 459.879,Z 461.461,A -85,B 0,C 180,E1 -8002.979,E2 -8002.979} C_VEL
LIN {X 0,Y 459.731,Z 466.134,A -85,B 0,C 180,E1 -8003.859,E2 -8003.859} C_VEL
LIN {X 0,Y 459.71,Z 470.01,A -85,B 0,C 180,E1 -8004.739,E2 -8004.739} C_VEL
LIN {X 0,Y 459.6,Z 474.415,A -85,B 0,C 180,E1 -8006.056,E2 -8006.056} C_VEL
LIN {X 0,Y 459.593,Z 477.486,A -85,B 0,C 180,E1 -8007.372,E2 -8007.372} C_VEL
LIN {X 0,Y 459.545,Z 478.843,A -85,B 0,C 180,E1 -8008.249,E2 -8008.249} C_VEL
LIN {X 0,Y 459.554,Z 479.695,A -85,B 0,C 180,E1 -8009.125,E2 -8009.125} C_VEL
LIN {X 0,Y 459.534,Z 479.993,A -85,B 0,C 180,E1 -8010.001,E2 -8010.001} C_VEL
LIN {X 0,Y 459.525,Z 479.69,A -85,B 0,C 180,E1 -8010.878,E2 -8010.878} C_VEL
LIN {X 0,Y 459.545,Z 478.888,A -85,B 0,C 180,E1 -8011.754,E2 -8011.754} C_VEL
LIN {X 0,Y 459.594,Z 477.578,A -85,B 0,C 180,E1 -8012.631,E2 -8012.631} C_VEL
LIN {X 0,Y 459.588,Z 474.531,A -85,B 0,C 180,E1 -8013.947,E2 -8013.947} C_VEL
LIN {X 0,Y 459.651,Z 471.755,A -85,B 0,C 180,E1 -8014.825,E2 -8014.825} C_VEL
LIN {X 0,Y 459.747,Z 468.327,A -85,B 0,C 180,E1 -8015.704,E2 -8015.704} C_VEL
LIN {X 0,Y 459.842,Z 463.149,A -85,B 0,C 180,E1 -8016.766,E2 -8016.766} C_VEL
LIN {X 0,Y 460.011,Z 457.669,A -85,B 0,C 180,E1 -8017.684,E2 -8017.684} C_VEL
LIN {X 0,Y 460.193,Z 451.317,A -85,B 0,C 180,E1 -8018.565,E2 -8018.565} C_VEL
LIN {X 0,Y 460.418,Z 444.663,A -85,B 0,C 180,E1 -8019.335,E2 -8019.335} C_VEL
LIN {X 0,Y 460.746,Z 436.638,A -85,B 0,C 180,E1 -8020.104,E2 -8020.104} C_VEL
LIN {X 0,Y 461.1,Z 426.669,A -85,B 0,C 180,E1 -8020.873,E2 -8020.873} C_VEL
LIN {X 0,Y 461.466,Z 416.236,A -85,B 0,C 180,E1 -8021.476,E2 -8021.476} C_VEL
LIN {X 0,Y 461.722,Z 405.806,A -85,B 0,C 180,E1 -8021.915,E2 -8021.915} C_VEL
LIN {X 0,Y 461.963,Z 396.381,A -85,B 0,C 180,E1 -8022.187,E2 -8022.187} C_VEL
LIN {X 0,Y 462.594,Z 335.365,A -85,B 0,C 180,E1 -8023.325,E2 -8023.325} C_VEL
LIN {X 0,Y 460.415,Z 318.13,A -85,B 0,C 180,E1 -8023.743,E2 -8023.743} C_VEL
LIN {X 0,Y 460.802,Z 298.556,A -85,B 0,C 180,E1 -8027.303,E2 -8027.303} C_VEL
LIN {X 0,Y 461.11,Z 280.638,A -85,B 0,C 180,E1 -8030.522,E2 -8030.522} C_VEL
LIN {X 0,Y 461.141,Z 271.484,A -85,B 0,C 180,E1 -8032.174,E2 -8032.174} C_VEL
LIN {X 0,Y 460.593,Z 267.929,A -85,B 0,C 180,E1 -8032.84,E2 -8032.84} C_VEL
LIN {X 0,Y 460.482,Z 267.94,A -85,B 0,C 180,E1 -8036.272,E2 -8036.272} C_VEL
LIN {X 0,Y 460.509,Z 267.938,A -85,B 0,C 180,E1 -8039.234,E2 -8039.234} C_VEL
LIN {X 0,Y 460.492,Z 267.936,A -85,B 0,C 180,E1 -8042.289,E2 -8042.289} C_VEL
LIN {X 0,Y 460.459,Z 267.94,A -85,B 0,C 180,E1 -8045.451,E2 -8045.451} C_VEL
LIN {X 0,Y 460.505,Z 267.936,A -85,B 0,C 180,E1 -8048.736,E2 -8048.736} C_VEL
LIN {X 0,Y 460.509,Z 267.931,A -85,B 0,C 180,E1 -8051.596,E2 -8051.596} C_VEL
LIN {X 0,Y 460.508,Z 267.934,A -85,B 0,C 180,E1 -8054.591,E2 -8054.591} C_VEL
LIN {X 0,Y 460.489,Z 267.932,A -85,B 0,C 180,E1 -8057.812,E2 -8057.812} C_VEL
LIN {X 0,Y 460.525,Z 267.926,A -85,B 0,C 180,E1 -8060.134,E2 -8060.134} C_VEL
LIN {X 0,Y 460.485,Z 267.935,A -85,B 0,C 180,E1 -8063.468,E2 -8063.468} C_VEL
LIN {X 0,Y 460.532,Z 267.931,A -85,B 0,C 180,E1 -8066.672,E2 -8066.672} C_VEL
LIN {X 0,Y 460.52,Z 267.932,A -85,B 0,C 180,E1 -8069.758,E2 -8069.758} C_VEL
LIN {X 0,Y 460.53,Z 267.933,A -85,B 0,C 180,E1 -8072.75,E2 -8072.75} C_VEL
LIN {X 0,Y 460.537,Z 267.933,A -85,B 0,C 180,E1 -8075.664,E2 -8075.664} C_VEL
LIN {X 0,Y 460.536,Z 267.933,A -85,B 0,C 180,E1 -8078.576,E2 -8078.576} C_VEL
LIN {X 0,Y 460.601,Z 267.927,A -85,B 0,C 180,E1 -8081.308,E2 -8081.308} C_VEL
LIN {X 0,Y 460.72,Z 267.979,A -85,B 0,C 180,E1 -8083.778,E2 -8083.778} C_VEL
LIN {X 0,Y 460.993,Z 271.526,A -85,B 0,C 180,E1 -8084.296,E2 -8084.296} C_VEL
LIN {X 0,Y 460.757,Z 285.15,A -85,B 0,C 180,E1 -8086.278,E2 -8086.278} C_VEL
LIN {X 0,Y 462.937,Z 300.096,A -85,B 0,C 180,E1 -8086.664,E2 -8086.664} C_VEL
LIN {X 0,Y 462.082,Z 365.538,A -85,B 0,C 180,E1 -8087.897,E2 -8087.897} C_VEL
LIN {X 0,Y 461.831,Z 377.969,A -85,B 0,C 180,E1 -8088.308,E2 -8088.308} C_VEL
LIN {X 0,Y 461.585,Z 387.855,A -85,B 0,C 180,E1 -8088.802,E2 -8088.802} C_VEL
LIN {X 0,Y 461.321,Z 396.366,A -85,B 0,C 180,E1 -8089.351,E2 -8089.351} C_VEL
LIN {X 0,Y 461.129,Z 404.556,A -85,B 0,C 180,E1 -8090.013,E2 -8090.013} C_VEL
LIN {X 0,Y 460.859,Z 412.351,A -85,B 0,C 180,E1 -8090.782,E2 -8090.782} C_VEL
LIN {X 0,Y 460.555,Z 419.649,A -85,B 0,C 180,E1 -8091.661,E2 -8091.661} C_VEL
LIN {X 0,Y 460.243,Z 427.03,A -85,B 0,C 180,E1 -8092.759,E2 -8092.759} C_VEL
LIN {X 0,Y 460.131,Z 432.775,A -85,B 0,C 180,E1 -8093.858,E2 -8093.858} C_VEL
LIN {X 0,Y 459.813,Z 436.572,A -85,B 0,C 180,E1 -8094.734,E2 -8094.734} C_VEL
LIN {X 0,Y 459.889,Z 439.629,A -85,B 0,C 180,E1 -8095.614,E2 -8095.614} C_VEL
LIN {X 0,Y 459.78,Z 442.011,A -85,B 0,C 180,E1 -8096.49,E2 -8096.49} C_VEL
LIN {X 0,Y 459.669,Z 443.82,A -85,B 0,C 180,E1 -8097.367,E2 -8097.367} C_VEL
LIN {X 0,Y 459.608,Z 445.105,A -85,B 0,C 180,E1 -8098.243,E2 -8098.243} C_VEL
LIN {X 0,Y 459.558,Z 445.891,A -85,B 0,C 180,E1 -8099.119,E2 -8099.119} C_VEL
LIN {X 0,Y 459.536,Z 446.161,A -85,B 0,C 180,E1 -8099.996,E2 -8099.996} C_VEL
LIN {X 0,Y 459.557,Z 445.824,A -85,B 0,C 180,E1 -8100.872,E2 -8100.872} C_VEL
LIN {X 0,Y 459.577,Z 444.97,A -85,B 0,C 180,E1 -8101.748,E2 -8101.748} C_VEL
LIN {X 0,Y 459.646,Z 443.616,A -85,B 0,C 180,E1 -8102.625,E2 -8102.625} C_VEL
LIN {X 0,Y 459.797,Z 440.537,A -85,B 0,C 180,E1 -8103.939,E2 -8103.939} C_VEL
LIN {X 0,Y 459.79,Z 436.15,A -85,B 0,C 180,E1 -8105.257,E2 -8105.257} C_VEL
LIN {X 0,Y 460.152,Z 430.138,A -85,B 0,C 180,E1 -8106.558,E2 -8106.558} C_VEL
LIN {X 0,Y 460.195,Z 424.987,A -85,B 0,C 180,E1 -8107.454,E2 -8107.454} C_VEL
LIN {X 0,Y 460.402,Z 418.863,A -85,B 0,C 180,E1 -8108.333,E2 -8108.333} C_VEL
LIN {X 0,Y 460.659,Z 411.412,A -85,B 0,C 180,E1 -8109.213,E2 -8109.213} C_VEL
LIN {X 0,Y 460.944,Z 403.445,A -85,B 0,C 180,E1 -8109.983,E2 -8109.983} C_VEL
LIN {X 0,Y 461.26,Z 393.53,A -85,B 0,C 180,E1 -8110.752,E2 -8110.752} C_VEL
LIN {X 0,Y 461.535,Z 381.954,A -85,B 0,C 180,E1 -8111.412,E2 -8111.412} C_VEL
LIN {X 0,Y 461.729,Z 372.703,A -85,B 0,C 180,E1 -8111.797,E2 -8111.797} C_VEL
LIN {X 0,Y 461.873,Z 363.203,A -85,B 0,C 180,E1 -8112.072,E2 -8112.072} C_VEL
LIN {X 0,Y 462.316,Z 298.867,A -85,B 0,C 180,E1 -8113.235,E2 -8113.235} C_VEL
LIN {X 0,Y 460.476,Z 287.295,A -85,B 0,C 180,E1 -8113.507,E2 -8113.507} C_VEL
LIN {X 0,Y 460.786,Z 274.136,A -85,B 0,C 180,E1 -8116.84,E2 -8116.84} C_VEL
LIN {X 0,Y 460.637,Z 267.921,A -85,B 0,C 180,E1 -8118.48,E2 -8118.48} C_VEL
LIN {X 0,Y 460.504,Z 267.936,A -85,B 0,C 180,E1 -8121.48,E2 -8121.48} C_VEL
LIN {X 0,Y 460.503,Z 267.934,A -85,B 0,C 180,E1 -8124.328,E2 -8124.328} C_VEL
LIN {X 0,Y 460.474,Z 267.939,A -85,B 0,C 180,E1 -8127.244,E2 -8127.244} C_VEL
LIN {X 0,Y 460.482,Z 267.936,A -85,B 0,C 180,E1 -8130.235,E2 -8130.235} C_VEL
LIN {X 0,Y 460.505,Z 267.936,A -85,B 0,C 180,E1 -8133.319,E2 -8133.319} C_VEL
LIN {X 0,Y 460.446,Z 267.94,A -85,B 0,C 180,E1 -8136.524,E2 -8136.524} C_VEL
LIN {X 0,Y 460.489,Z 267.938,A -85,B 0,C 180,E1 -8139.858,E2 -8139.858} C_VEL
LIN {X 0,Y 460.46,Z 267.939,A -85,B 0,C 180,E1 -8142.892,E2 -8142.892} C_VEL
LIN {X 0,Y 460.472,Z 267.939,A -85,B 0,C 180,E1 -8145.826,E2 -8145.826} C_VEL
LIN {X 0,Y 460.493,Z 267.935,A -85,B 0,C 180,E1 -8148.983,E2 -8148.983} C_VEL
LIN {X 0,Y 460.479,Z 267.938,A -85,B 0,C 180,E1 -8151.261,E2 -8151.261} C_VEL
LIN {X 0,Y 460.471,Z 267.939,A -85,B 0,C 180,E1 -8154.55,E2 -8154.55} C_VEL
LIN {X 0,Y 460.487,Z 267.939,A -85,B 0,C 180,E1 -8157.711,E2 -8157.711} C_VEL
LIN {X 0,Y 460.494,Z 267.935,A -85,B 0,C 180,E1 -8160.765,E2 -8160.765} C_VEL
LIN {X 0,Y 460.517,Z 267.934,A -85,B 0,C 180,E1 -8163.731,E2 -8163.731} C_VEL
LIN {X 0,Y 460.49,Z 267.937,A -85,B 0,C 180,E1 -8166.504,E2 -8166.504} C_VEL
LIN {X 0,Y 459.845,Z 268.02,A -85,B 0,C 180,E1 -8167.234,E2 -8167.234} C_VEL
LIN {X 0,Y 456.992,Z 268.377,A -85,B 0,C 180,E1 -8168.42,E2 -8168.42} C_VEL
LIN {X 0,Y 454.566,Z 268.678,A -85,B 0,C 180,E1 -8169.376,E2 -8169.376} C_VEL
LIN {X 0,Y 453.526,Z 268.805,A -85,B 0,C 180,E1 -8170.116,E2 -8170.116} C_VEL
LIN {X 0,Y 453.444,Z 268.814,A -85,B 0,C 180,E1 -8170.366,E2 -8170.366} C_VEL
LIN {X 0,Y 453.514,Z 268.806,A -85,B 0,C 180,E1 -8173.876,E2 -8173.876} C_VEL
LIN {X 0,Y 453.547,Z 268.8,A -85,B 0,C 180,E1 -8177.469,E2 -8177.469} C_VEL
LIN {X 0,Y 453.537,Z 268.804,A -85,B 0,C 180,E1 -8181.084,E2 -8181.084} C_VEL
LIN {X 0,Y 453.624,Z 268.79,A -85,B 0,C 180,E1 -8183.773,E2 -8183.773} C_VEL
LIN {X 0,Y 453.715,Z 268.781,A -85,B 0,C 180,E1 -8187.335,E2 -8187.335} C_VEL
LIN {X 0,Y 453.762,Z 268.773,A -85,B 0,C 180,E1 -8189.998,E2 -8189.998} C_VEL
LIN {X 0,Y 453.714,Z 268.783,A -85,B 0,C 180,E1 -8192.662,E2 -8192.662} C_VEL
LIN {X 0,Y 453.622,Z 268.791,A -85,B 0,C 180,E1 -8196.224,E2 -8196.224} C_VEL
LIN {X 0,Y 453.538,Z 268.804,A -85,B 0,C 180,E1 -8198.913,E2 -8198.913} C_VEL
LIN {X 0,Y 453.541,Z 268.802,A -85,B 0,C 180,E1 -8202.551,E2 -8202.551} C_VEL
LIN {X 0,Y 453.484,Z 268.808,A -85,B 0,C 180,E1 -8206.196,E2 -8206.196} C_VEL
LIN {X 0,Y 453.459,Z 268.814,A -85,B 0,C 180,E1 -8209.041,E2 -8209.041} C_VEL
LIN {X 0,Y 453.418,Z 268.818,A -85,B 0,C 180,E1 -8211.837,E2 -8211.837} C_VEL
LIN {X 0,Y 453.466,Z 268.81,A -85,B 0,C 180,E1 -8214.735,E2 -8214.735} C_VEL
LIN {X 0,Y 453.48,Z 268.81,A -85,B 0,C 180,E1 -8217.963,E2 -8217.963} C_VEL
LIN {X 0,Y 453.426,Z 268.815,A -85,B 0,C 180,E1 -8220.761,E2 -8220.761} C_VEL
LIN {X 0,Y 453.422,Z 268.817,A -85,B 0,C 180,E1 -8223.915,E2 -8223.915} C_VEL
LIN {X 0,Y 453.418,Z 268.817,A -85,B 0,C 180,E1 -8227.19,E2 -8227.19} C_VEL
LIN {X 0,Y 453.486,Z 268.81,A -85,B 0,C 180,E1 -8229.448,E2 -8229.448} C_VEL
LIN {X 0,Y 453.441,Z 268.813,A -85,B 0,C 180,E1 -8232.995,E2 -8232.995} C_VEL
LIN {X 0,Y 453.427,Z 268.819,A -85,B 0,C 180,E1 -8235.784,E2 -8235.784} C_VEL
LIN {X 0,Y 453.449,Z 268.814,A -85,B 0,C 180,E1 -8238.215,E2 -8238.215} C_VEL
LIN {X 0,Y 453.484,Z 268.81,A -85,B 0,C 180,E1 -8240.792,E2 -8240.792} C_VEL
LIN {X 0,Y 453.413,Z 268.82,A -85,B 0,C 180,E1 -8243.921,E2 -8243.921} C_VEL
LIN {X 0,Y 453.442,Z 268.814,A -85,B 0,C 180,E1 -8247.155,E2 -8247.155} C_VEL
LIN {X 0,Y 453.435,Z 268.817,A -85,B 0,C 180,E1 -8250.272,E2 -8250.272} C_VEL
LIN {X 0,Y 453.451,Z 268.813,A -85,B 0,C 180,E1 -8253.297,E2 -8253.297} C_VEL
LIN {X 0,Y 453.459,Z 268.814,A -85,B 0,C 180,E1 -8256.243,E2 -8256.243} C_VEL
LIN {X 0,Y 453.449,Z 268.814,A -85,B 0,C 180,E1 -8259.122,E2 -8259.122} C_VEL
LIN {X 0,Y 453.471,Z 268.809,A -85,B 0,C 180,E1 -8261.949,E2 -8261.949} C_VEL
LIN {X 0,Y 453.51,Z 268.807,A -85,B 0,C 180,E1 -8264.731,E2 -8264.731} C_VEL
LIN {X 0,Y 453.532,Z 268.803,A -85,B 0,C 180,E1 -8268.383,E2 -8268.383} C_VEL
LIN {X 0,Y 453.56,Z 268.8,A -85,B 0,C 180,E1 -8271.091,E2 -8271.091} C_VEL
LIN {X 0,Y 453.637,Z 268.79,A -85,B 0,C 180,E1 -8273.779,E2 -8273.779} C_VEL
LIN {X 0,Y 453.692,Z 268.784,A -85,B 0,C 180,E1 -8277.341,E2 -8277.341} C_VEL
LIN {X 0,Y 453.771,Z 268.773,A -85,B 0,C 180,E1 -8280.004,E2 -8280.004} C_VEL
LIN {X 0,Y 453.716,Z 268.779,A -85,B 0,C 180,E1 -8282.668,E2 -8282.668} C_VEL
LIN {X 0,Y 453.628,Z 268.79,A -85,B 0,C 180,E1 -8286.23,E2 -8286.23} C_VEL
LIN {X 0,Y 453.57,Z 268.798,A -85,B 0,C 180,E1 -8288.918,E2 -8288.918} C_VEL
LIN {X 0,Y 453.553,Z 268.799,A -85,B 0,C 180,E1 -8292.533,E2 -8292.533} C_VEL
LIN {X 0,Y 453.493,Z 268.809,A -85,B 0,C 180,E1 -8296.095,E2 -8296.095} C_VEL
LIN {X 0,Y 453.508,Z 268.805,A -85,B 0,C 180,E1 -8299.043,E2 -8299.043} C_VEL
LIN {X 0,Y 453.468,Z 268.812,A -85,B 0,C 180,E1 -8301.84,E2 -8301.84} C_VEL
LIN {X 0,Y 453.463,Z 268.811,A -85,B 0,C 180,E1 -8304.741,E2 -8304.741} C_VEL
LIN {X 0,Y 453.484,Z 268.81,A -85,B 0,C 180,E1 -8307.953,E2 -8307.953} C_VEL
LIN {X 0,Y 453.471,Z 268.811,A -85,B 0,C 180,E1 -8310.763,E2 -8310.763} C_VEL
LIN {X 0,Y 453.462,Z 268.815,A -85,B 0,C 180,E1 -8313.917,E2 -8313.917} C_VEL
LIN {X 0,Y 453.435,Z 268.814,A -85,B 0,C 180,E1 -8317.194,E2 -8317.194} C_VEL
LIN {X 0,Y 453.468,Z 268.811,A -85,B 0,C 180,E1 -8320.615,E2 -8320.615} C_VEL
LIN {X 0,Y 453.456,Z 268.815,A -85,B 0,C 180,E1 -8324.225,E2 -8324.225} C_VEL
LIN {X 0,Y 453.415,Z 268.818,A -85,B 0,C 180,E1 -8327.002,E2 -8327.002} C_VEL
LIN {X 0,Y 453.471,Z 268.81,A -85,B 0,C 180,E1 -8329.416,E2 -8329.416} C_VEL
LIN {X 0,Y 453.446,Z 268.814,A -85,B 0,C 180,E1 -8332.812,E2 -8332.812} C_VEL
LIN {X 0,Y 453.467,Z 268.81,A -85,B 0,C 180,E1 -8336.089,E2 -8336.089} C_VEL
LIN {X 0,Y 453.456,Z 268.813,A -85,B 0,C 180,E1 -8339.241,E2 -8339.241} C_VEL
LIN {X 0,Y 453.474,Z 268.81,A -85,B 0,C 180,E1 -8342.296,E2 -8342.296} C_VEL
LIN {X 0,Y 453.533,Z 268.912,A -85,B 0,C 180,E1 -8345.612,E2 -8345.612} C_VEL
LIN {X 0,Y 454.994,Z 278.243,A -85,B 0,C 180,E1 -8347.68,E2 -8347.68} C_VEL
LIN {X 0,Y 454.423,Z 292.335,A -85,B 0,C 180,E1 -8350.637,E2 -8350.637} C_VEL
LIN {X 0,Y 453.758,Z 308.233,A -85,B 0,C 180,E1 -8353.932,E2 -8353.932} C_VEL
LIN {X 0,Y 453.385,Z 319.91,A -85,B 0,C 180,E1 -8356.328,E2 -8356.328} C_VEL
LIN {X 0,Y 455.394,Z 337.683,A -85,B 0,C 180,E1 -8356.717,E2 -8356.717} C_VEL
LIN {X 0,Y 454.786,Z 397.54,A -85,B 0,C 180,E1 -8357.819,E2 -8357.819} C_VEL
LIN {X 0,Y 454.495,Z 408.363,A -85,B 0,C 180,E1 -8358.15,E2 -8358.15} C_VEL
LIN {X 0,Y 454.158,Z 420.608,A -85,B 0,C 180,E1 -8358.735,E2 -8358.735} C_VEL
LIN {X 0,Y 453.847,Z 429.25,A -85,B 0,C 180,E1 -8359.292,E2 -8359.292} C_VEL
LIN {X 0,Y 453.634,Z 437.571,A -85,B 0,C 180,E1 -8359.964,E2 -8359.964} C_VEL
LIN {X 0,Y 453.285,Z 445.465,A -85,B 0,C 180,E1 -8360.745,E2 -8360.745} C_VEL
LIN {X 0,Y 453.084,Z 452.004,A -85,B 0,C 180,E1 -8361.528,E2 -8361.528} C_VEL
LIN {X 0,Y 452.88,Z 459.685,A -85,B 0,C 180,E1 -8362.646,E2 -8362.646} C_VEL
LIN {X 0,Y 452.659,Z 465.703,A -85,B 0,C 180,E1 -8363.762,E2 -8363.762} C_VEL
LIN {X 0,Y 452.623,Z 469.605,A -85,B 0,C 180,E1 -8364.656,E2 -8364.656} C_VEL
LIN {X 0,Y 452.5,Z 474.061,A -85,B 0,C 180,E1 -8365.994,E2 -8365.994} C_VEL
LIN {X 0,Y 452.518,Z 477.165,A -85,B 0,C 180,E1 -8367.331,E2 -8367.331} C_VEL
LIN {X 0,Y 452.46,Z 478.546,A -85,B 0,C 180,E1 -8368.221,E2 -8368.221} C_VEL
LIN {X 0,Y 452.459,Z 479.419,A -85,B 0,C 180,E1 -8369.112,E2 -8369.112} C_VEL
LIN {X 0,Y 452.468,Z 479.722,A -85,B 0,C 180,E1 -8370.002,E2 -8370.002} C_VEL
LIN {X 0,Y 452.432,Z 479.429,A -85,B 0,C 180,E1 -8370.892,E2 -8370.892} C_VEL
LIN {X 0,Y 452.46,Z 478.637,A -85,B 0,C 180,E1 -8371.782,E2 -8371.782} C_VEL
LIN {X 0,Y 452.518,Z 477.338,A -85,B 0,C 180,E1 -8372.672,E2 -8372.672} C_VEL
LIN {X 0,Y 452.491,Z 474.29,A -85,B 0,C 180,E1 -8374.009,E2 -8374.009} C_VEL
LIN {X 0,Y 452.583,Z 471.522,A -85,B 0,C 180,E1 -8374.901,E2 -8374.901} C_VEL
LIN {X 0,Y 452.661,Z 466.12,A -85,B 0,C 180,E1 -8376.241,E2 -8376.241} C_VEL
LIN {X 0,Y 452.905,Z 458.964,A -85,B 0,C 180,E1 -8377.581,E2 -8377.581} C_VEL
LIN {X 0,Y 453.101,Z 452.938,A -85,B 0,C 180,E1 -8378.475,E2 -8378.475} C_VEL
LIN {X 0,Y 453.379,Z 445.614,A -85,B 0,C 180,E1 -8379.369,E2 -8379.369} C_VEL
LIN {X 0,Y 453.715,Z 437.821,A -85,B 0,C 180,E1 -8380.15,E2 -8380.15} C_VEL
LIN {X 0,Y 454.012,Z 429.669,A -85,B 0,C 180,E1 -8380.819,E2 -8380.819} C_VEL
LIN {X 0,Y 454.306,Z 421.273,A -85,B 0,C 180,E1 -8381.377,E2 -8381.377} C_VEL
LIN {X 0,Y 454.642,Z 411.605,A -85,B 0,C 180,E1 -8381.877,E2 -8381.877} C_VEL
LIN {X 0,Y 455.016,Z 399.387,A -85,B 0,C 180,E1 -8382.32,E2 -8382.32} C_VEL
LIN {X 0,Y 455.342,Z 375.026,A -85,B 0,C 180,E1 -8382.803,E2 -8382.803} C_VEL
LIN {X 0,Y 455.739,Z 335.854,A -85,B 0,C 180,E1 -8383.556,E2 -8383.556} C_VEL
LIN {X 0,Y 453.372,Z 317.818,A -85,B 0,C 180,E1 -8384.018,E2 -8384.018} C_VEL
LIN {X 0,Y 453.782,Z 299.583,A -85,B 0,C 180,E1 -8387.347,E2 -8387.347} C_VEL
LIN {X 0,Y 454.144,Z 281.735,A -85,B 0,C 180,E1 -8390.615,E2 -8390.615} C_VEL
LIN {X 0,Y 454.171,Z 272.585,A -85,B 0,C 180,E1 -8392.28,E2 -8392.28} C_VEL
LIN {X 0,Y 453.549,Z 268.806,A -85,B 0,C 180,E1 -8393.034,E2 -8393.034} C_VEL
LIN {X 0,Y 453.47,Z 268.812,A -85,B 0,C 180,E1 -8395.983,E2 -8395.983} C_VEL
LIN {X 0,Y 453.459,Z 268.818,A -85,B 0,C 180,E1 -8398.717,E2 -8398.717} C_VEL
LIN {X 0,Y 453.432,Z 268.814,A -85,B 0,C 180,E1 -8401.803,E2 -8401.803} C_VEL
LIN {X 0,Y 453.415,Z 268.82,A -85,B 0,C 180,E1 -8404.996,E2 -8404.996} C_VEL
LIN {X 0,Y 453.451,Z 268.811,A -85,B 0,C 180,E1 -8408.314,E2 -8408.314} C_VEL
LIN {X 0,Y 453.479,Z 268.809,A -85,B 0,C 180,E1 -8410.612,E2 -8410.612} C_VEL
LIN {X 0,Y 453.453,Z 268.81,A -85,B 0,C 180,E1 -8414.224,E2 -8414.224} C_VEL
LIN {X 0,Y 453.431,Z 268.819,A -85,B 0,C 180,E1 -8416.998,E2 -8416.998} C_VEL
LIN {X 0,Y 453.486,Z 268.806,A -85,B 0,C 180,E1 -8419.412,E2 -8419.412} C_VEL
LIN {X 0,Y 453.461,Z 268.812,A -85,B 0,C 180,E1 -8422.808,E2 -8422.808} C_VEL
LIN {X 0,Y 453.482,Z 268.806,A -85,B 0,C 180,E1 -8426.085,E2 -8426.085} C_VEL
LIN {X 0,Y 453.49,Z 268.81,A -85,B 0,C 180,E1 -8429.238,E2 -8429.238} C_VEL
LIN {X 0,Y 453.506,Z 268.806,A -85,B 0,C 180,E1 -8432.292,E2 -8432.292} C_VEL
LIN {X 0,Y 453.509,Z 268.812,A -85,B 0,C 180,E1 -8435.262,E2 -8435.262} C_VEL
LIN {X 0,Y 453.495,Z 268.81,A -85,B 0,C 180,E1 -8438.412,E2 -8438.412} C_VEL
LIN {X 0,Y 453.537,Z 268.806,A -85,B 0,C 180,E1 -8441.006,E2 -8441.006} C_VEL
LIN {X 0,Y 453.667,Z 268.882,A -85,B 0,C 180,E1 -8443.571,E2 -8443.571} C_VEL
LIN {X 0,Y 454.123,Z 272.472,A -85,B 0,C 180,E1 -8444.114,E2 -8444.114} C_VEL
LIN {X 0,Y 453.882,Z 285.581,A -85,B 0,C 180,E1 -8446.013,E2 -8446.013} C_VEL
LIN {X 0,Y 456.131,Z 300.722,A -85,B 0,C 180,E1 -8446.415,E2 -8446.415} C_VEL
LIN {X 0,Y 455.186,Z 366.699,A -85,B 0,C 180,E1 -8447.711,E2 -8447.711} C_VEL
LIN {X 0,Y 454.915,Z 378.688,A -85,B 0,C 180,E1 -8448.128,E2 -8448.128} C_VEL
LIN {X 0,Y 454.669,Z 388.475,A -85,B 0,C 180,E1 -8448.63,E2 -8448.63} C_VEL
LIN {X 0,Y 454.385,Z 396.925,A -85,B 0,C 180,E1 -8449.187,E2 -8449.187} C_VEL
LIN {X 0,Y 454.162,Z 405.076,A -85,B 0,C 180,E1 -8449.858,E2 -8449.858} C_VEL
LIN {X 0,Y 453.89,Z 412.84,A -85,B 0,C 180,E1 -8450.639,E2 -8450.639} C_VEL
LIN {X 0,Y 453.461,Z 421.78,A -85,B 0,C 180,E1 -8451.754,E2 -8451.754} C_VEL
LIN {X 0,Y 453.204,Z 428.655,A -85,B 0,C 180,E1 -8452.869,E2 -8452.869} C_VEL
LIN {X 0,Y 453.102,Z 433.177,A -85,B 0,C 180,E1 -8453.763,E2 -8453.763} C_VEL
LIN {X 0,Y 452.762,Z 436.948,A -85,B 0,C 180,E1 -8454.652,E2 -8454.652} C_VEL
LIN {X 0,Y 452.816,Z 439.99,A -85,B 0,C 180,E1 -8455.545,E2 -8455.545} C_VEL
LIN {X 0,Y 452.719,Z 442.354,A -85,B 0,C 180,E1 -8456.436,E2 -8456.436} C_VEL
LIN {X 0,Y 452.593,Z 444.142,A -85,B 0,C 180,E1 -8457.326,E2 -8457.326} C_VEL
LIN {X 0,Y 452.52,Z 445.407,A -85,B 0,C 180,E1 -8458.216,E2 -8458.216} C_VEL
LIN {X 0,Y 452.464,Z 446.171,A -85,B 0,C 180,E1 -8459.106,E2 -8459.106} C_VEL
LIN {X 0,Y 452.47,Z 446.427,A -85,B 0,C 180,E1 -8459.996,E2 -8459.996} C_VEL
LIN {X 0,Y 452.463,Z 446.079,A -85,B 0,C 180,E1 -8460.885,E2 -8460.885} C_VEL
LIN {X 0,Y 452.491,Z 445.199,A -85,B 0,C 180,E1 -8461.776,E2 -8461.776} C_VEL
LIN {X 0,Y 452.572,Z 443.814,A -85,B 0,C 180,E1 -8462.666,E2 -8462.666} C_VEL
LIN {X 0,Y 452.726,Z 440.701,A -85,B 0,C 180,E1 -8464.001,E2 -8464.001} C_VEL
LIN {X 0,Y 452.736,Z 436.265,A -85,B 0,C 180,E1 -8465.34,E2 -8465.34} C_VEL
LIN {X 0,Y 453.075,Z 430.298,A -85,B 0,C 180,E1 -8466.638,E2 -8466.638} C_VEL
LIN {X 0,Y 453.148,Z 424.971,A -85,B 0,C 180,E1 -8467.57,E2 -8467.57} C_VEL
LIN {X 0,Y 453.354,Z 418.783,A -85,B 0,C 180,E1 -8468.464,E2 -8468.464} C_VEL
LIN {X 0,Y 453.652,Z 411.256,A -85,B 0,C 180,E1 -8469.357,E2 -8469.357} C_VEL
LIN {X 0,Y 453.945,Z 403.203,A -85,B 0,C 180,E1 -8470.138,E2 -8470.138} C_VEL
LIN {X 0,Y 454.274,Z 393.156,A -85,B 0,C 180,E1 -8470.919,E2 -8470.919} C_VEL
LIN {X 0,Y 454.53,Z 382.458,A -85,B 0,C 180,E1 -8471.534,E2 -8471.534} C_VEL
LIN {X 0,Y 454.71,Z 372.51,A -85,B 0,C 180,E1 -8471.953,E2 -8471.953} C_VEL
LIN {X 0,Y 454.896,Z 362.849,A -85,B 0,C 180,E1 -8472.231,E2 -8472.231} C_VEL
LIN {X 0,Y 455.375,Z 299.617,A -85,B 0,C 180,E1 -8473.396,E2 -8473.396} C_VEL
LIN {X 0,Y 453.433,Z 287.483,A -85,B 0,C 180,E1 -8473.695,E2 -8473.695} C_VEL
LIN {X 0,Y 453.788,Z 274.179,A -85,B 0,C 180,E1 -8477.108,E2 -8477.108} C_VEL
LIN {X 0,Y 453.58,Z 268.8,A -85,B 0,C 180,E1 -8478.573,E2 -8478.573} C_VEL
LIN {X 0,Y 453.464,Z 268.811,A -85,B 0,C 180,E1 -8481.831,E2 -8481.831} C_VEL
LIN {X 0,Y 453.472,Z 268.813,A -85,B 0,C 180,E1 -8484.73,E2 -8484.73} C_VEL
LIN {X 0,Y 453.445,Z 268.813,A -85,B 0,C 180,E1 -8487.937,E2 -8487.937} C_VEL
LIN {X 0,Y 453.436,Z 268.816,A -85,B 0,C 180,E1 -8490.755,E2 -8490.755} C_VEL
LIN {X 0,Y 453.452,Z 268.814,A -85,B 0,C 180,E1 -8493.907,E2 -8493.907} C_VEL
LIN {X 0,Y 453.423,Z 268.818,A -85,B 0,C 180,E1 -8497.184,E2 -8497.184} C_VEL
LIN {X 0,Y 453.464,Z 268.81,A -85,B 0,C 180,E1 -8500.603,E2 -8500.603} C_VEL
LIN {X 0,Y 453.427,Z 268.817,A -85,B 0,C 180,E1 -8504.216,E2 -8504.216} C_VEL
LIN {X 0,Y 453.426,Z 268.816,A -85,B 0,C 180,E1 -8506.999,E2 -8506.999} C_VEL
LIN {X 0,Y 453.457,Z 268.814,A -85,B 0,C 180,E1 -8509.404,E2 -8509.404} C_VEL
LIN {X 0,Y 453.413,Z 268.817,A -85,B 0,C 180,E1 -8512.805,E2 -8512.805} C_VEL
LIN {X 0,Y 453.435,Z 268.816,A -85,B 0,C 180,E1 -8516.082,E2 -8516.082} C_VEL
LIN {X 0,Y 453.431,Z 268.815,A -85,B 0,C 180,E1 -8519.236,E2 -8519.236} C_VEL
LIN {X 0,Y 453.496,Z 268.808,A -85,B 0,C 180,E1 -8522.294,E2 -8522.294} C_VEL
LIN {X 0,Y 453.465,Z 268.81,A -85,B 0,C 180,E1 -8525.261,E2 -8525.261} C_VEL
LIN {X 0,Y 453.429,Z 268.817,A -85,B 0,C 180,E1 -8528.411,E2 -8528.411} C_VEL
LIN {X 0,Y 453.444,Z 268.814,A -85,B 0,C 180,E1 -8530.366,E2 -8530.366} C_VEL
LIN {X 0,Y 452.781,Z 268.897,A -85,B 0,C 180,E1 -8531.107,E2 -8531.107} C_VEL
LIN {X 0,Y 449.93,Z 269.253,A -85,B 0,C 180,E1 -8532.311,E2 -8532.311} C_VEL
LIN {X 0,Y 447.528,Z 269.55,A -85,B 0,C 180,E1 -8533.283,E2 -8533.283} C_VEL
LIN {X 0,Y 446.516,Z 269.679,A -85,B 0,C 180,E1 -8534.033,E2 -8534.033} C_VEL
LIN {X 0,Y 446.443,Z 269.686,A -85,B 0,C 180,E1 -8534.287,E2 -8534.287} C_VEL
LIN {X 0,Y 446.498,Z 269.679,A -85,B 0,C 180,E1 -8537.359,E2 -8537.359} C_VEL
LIN {X 0,Y 446.483,Z 269.682,A -85,B 0,C 180,E1 -8540.942,E2 -8540.942} C_VEL
LIN {X 0,Y 446.592,Z 269.666,A -85,B 0,C 180,E1 -8543.674,E2 -8543.674} C_VEL
LIN {X 0,Y 446.659,Z 269.661,A -85,B 0,C 180,E1 -8547.293,E2 -8547.293} C_VEL
LIN {X 0,Y 446.733,Z 269.649,A -85,B 0,C 180,E1 -8549.998,E2 -8549.998} C_VEL
LIN {X 0,Y 446.658,Z 269.661,A -85,B 0,C 180,E1 -8552.704,E2 -8552.704} C_VEL
LIN {X 0,Y 446.591,Z 269.667,A -85,B 0,C 180,E1 -8556.323,E2 -8556.323} C_VEL
LIN {X 0,Y 446.484,Z 269.682,A -85,B 0,C 180,E1 -8559.055,E2 -8559.055} C_VEL
LIN {X 0,Y 446.474,Z 269.683,A -85,B 0,C 180,E1 -8562.729,E2 -8562.729} C_VEL
LIN {X 0,Y 446.43,Z 269.687,A -85,B 0,C 180,E1 -8566.459,E2 -8566.459} C_VEL
LIN {X 0,Y 446.409,Z 269.691,A -85,B 0,C 180,E1 -8569.304,E2 -8569.304} C_VEL
LIN {X 0,Y 446.36,Z 269.696,A -85,B 0,C 180,E1 -8572.201,E2 -8572.201} C_VEL
LIN {X 0,Y 446.413,Z 269.692,A -85,B 0,C 180,E1 -8575.153,E2 -8575.153} C_VEL
LIN {X 0,Y 446.427,Z 269.689,A -85,B 0,C 180,E1 -8578.18,E2 -8578.18} C_VEL
LIN {X 0,Y 446.363,Z 269.698,A -85,B 0,C 180,E1 -8581.302,E2 -8581.302} C_VEL
LIN {X 0,Y 446.375,Z 269.694,A -85,B 0,C 180,E1 -8584.525,E2 -8584.525} C_VEL
LIN {X 0,Y 446.387,Z 269.693,A -85,B 0,C 180,E1 -8588.086,E2 -8588.086} C_VEL
LIN {X 0,Y 446.396,Z 269.691,A -85,B 0,C 180,E1 -8590.924,E2 -8590.924} C_VEL
LIN {X 0,Y 446.395,Z 269.694,A -85,B 0,C 180,E1 -8593.844,E2 -8593.844} C_VEL
LIN {X 0,Y 446.398,Z 269.692,A -85,B 0,C 180,E1 -8596.4,E2 -8596.4} C_VEL
LIN {X 0,Y 446.422,Z 269.691,A -85,B 0,C 180,E1 -8599.809,E2 -8599.809} C_VEL
LIN {X 0,Y 446.388,Z 269.694,A -85,B 0,C 180,E1 -8602.127,E2 -8602.127} C_VEL
LIN {X 0,Y 446.388,Z 269.692,A -85,B 0,C 180,E1 -8605.481,E2 -8605.481} C_VEL
LIN {X 0,Y 446.376,Z 269.695,A -85,B 0,C 180,E1 -8608.704,E2 -8608.704} C_VEL
LIN {X 0,Y 446.447,Z 269.685,A -85,B 0,C 180,E1 -8611.826,E2 -8611.826} C_VEL
LIN {X 0,Y 446.403,Z 269.691,A -85,B 0,C 180,E1 -8614.851,E2 -8614.851} C_VEL
LIN {X 0,Y 446.415,Z 269.691,A -85,B 0,C 180,E1 -8618.25,E2 -8618.25} C_VEL
LIN {X 0,Y 446.42,Z 269.688,A -85,B 0,C 180,E1 -8621.653,E2 -8621.653} C_VEL
LIN {X 0,Y 446.478,Z 269.684,A -85,B 0,C 180,E1 -8624.484,E2 -8624.484} C_VEL
LIN {X 0,Y 446.49,Z 269.679,A -85,B 0,C 180,E1 -8628.198,E2 -8628.198} C_VEL
LIN {X 0,Y 446.507,Z 269.679,A -85,B 0,C 180,E1 -8630.949,E2 -8630.949} C_VEL
LIN {X 0,Y 446.606,Z 269.667,A -85,B 0,C 180,E1 -8633.681,E2 -8633.681} C_VEL
LIN {X 0,Y 446.642,Z 269.662,A -85,B 0,C 180,E1 -8637.299,E2 -8637.299} C_VEL
LIN {X 0,Y 446.72,Z 269.651,A -85,B 0,C 180,E1 -8640.005,E2 -8640.005} C_VEL
LIN {X 0,Y 446.663,Z 269.658,A -85,B 0,C 180,E1 -8642.71,E2 -8642.71} C_VEL
LIN {X 0,Y 446.597,Z 269.666,A -85,B 0,C 180,E1 -8646.329,E2 -8646.329} C_VEL
LIN {X 0,Y 446.517,Z 269.678,A -85,B 0,C 180,E1 -8649.06,E2 -8649.06} C_VEL
LIN {X 0,Y 446.511,Z 269.677,A -85,B 0,C 180,E1 -8652.734,E2 -8652.734} C_VEL
LIN {X 0,Y 446.444,Z 269.687,A -85,B 0,C 180,E1 -8656.213,E2 -8656.213} C_VEL
LIN {X 0,Y 446.46,Z 269.685,A -85,B 0,C 180,E1 -8659.307,E2 -8659.307} C_VEL
LIN {X 0,Y 446.409,Z 269.691,A -85,B 0,C 180,E1 -8662.204,E2 -8662.204} C_VEL
LIN {X 0,Y 446.415,Z 269.689,A -85,B 0,C 180,E1 -8665.158,E2 -8665.158} C_VEL
LIN {X 0,Y 446.435,Z 269.687,A -85,B 0,C 180,E1 -8668.185,E2 -8668.185} C_VEL
LIN {X 0,Y 446.41,Z 269.689,A -85,B 0,C 180,E1 -8671.304,E2 -8671.304} C_VEL
LIN {X 0,Y 446.417,Z 269.69,A -85,B 0,C 180,E1 -8674.527,E2 -8674.527} C_VEL
LIN {X 0,Y 446.396,Z 269.694,A -85,B 0,C 180,E1 -8678.08,E2 -8678.08} C_VEL
LIN {X 0,Y 446.399,Z 269.69,A -85,B 0,C 180,E1 -8681.397,E2 -8681.397} C_VEL
LIN {X 0,Y 446.418,Z 269.69,A -85,B 0,C 180,E1 -8684.895,E2 -8684.895} C_VEL
LIN {X 0,Y 446.399,Z 269.692,A -85,B 0,C 180,E1 -8688.608,E2 -8688.608} C_VEL
LIN {X 0,Y 446.407,Z 269.69,A -85,B 0,C 180,E1 -8691.925,E2 -8691.925} C_VEL
LIN {X 0,Y 446.422,Z 269.689,A -85,B 0,C 180,E1 -8695.479,E2 -8695.479} C_VEL
LIN {X 0,Y 446.409,Z 269.692,A -85,B 0,C 180,E1 -8698.701,E2 -8698.701} C_VEL
LIN {X 0,Y 446.409,Z 269.689,A -85,B 0,C 180,E1 -8701.843,E2 -8701.843} C_VEL
LIN {X 0,Y 446.486,Z 269.743,A -85,B 0,C 180,E1 -8705.468,E2 -8705.468} C_VEL
LIN {X 0,Y 447.888,Z 278.249,A -85,B 0,C 180,E1 -8707.391,E2 -8707.391} C_VEL
LIN {X 0,Y 447.703,Z 286.101,A -85,B 0,C 180,E1 -8709.078,E2 -8709.078} C_VEL
LIN {X 0,Y 447.02,Z 300.618,A -85,B 0,C 180,E1 -8712.149,E2 -8712.149} C_VEL
LIN {X 0,Y 446.417,Z 317.313,A -85,B 0,C 180,E1 -8715.645,E2 -8715.645} C_VEL
LIN {X 0,Y 446.336,Z 319.671,A -85,B 0,C 180,E1 -8716.137,E2 -8716.137} C_VEL
LIN {X 0,Y 448.421,Z 339.12,A -85,B 0,C 180,E1 -8716.57,E2 -8716.57} C_VEL
LIN {X 0,Y 447.782,Z 397.841,A -85,B 0,C 180,E1 -8717.683,E2 -8717.683} C_VEL
LIN {X 0,Y 447.502,Z 409.222,A -85,B 0,C 180,E1 -8718.049,E2 -8718.049} C_VEL
LIN {X 0,Y 447.189,Z 419.614,A -85,B 0,C 180,E1 -8718.558,E2 -8718.558} C_VEL
LIN {X 0,Y 446.862,Z 428.396,A -85,B 0,C 180,E1 -8719.123,E2 -8719.123} C_VEL
LIN {X 0,Y 446.611,Z 436.826,A -85,B 0,C 180,E1 -8719.805,E2 -8719.805} C_VEL
LIN {X 0,Y 446.275,Z 444.809,A -85,B 0,C 180,E1 -8720.598,E2 -8720.598} C_VEL
LIN {X 0,Y 446.04,Z 451.419,A -85,B 0,C 180,E1 -8721.393,E2 -8721.393} C_VEL
LIN {X 0,Y 445.822,Z 457.707,A -85,B 0,C 180,E1 -8722.301,E2 -8722.301} C_VEL
LIN {X 0,Y 445.661,Z 462.92,A -85,B 0,C 180,E1 -8723.21,E2 -8723.21} C_VEL
LIN {X 0,Y 445.528,Z 467.238,A -85,B 0,C 180,E1 -8724.116,E2 -8724.116} C_VEL
LIN {X 0,Y 445.512,Z 470.808,A -85,B 0,C 180,E1 -8725.024,E2 -8725.024} C_VEL
LIN {X 0,Y 445.421,Z 474.891,A -85,B 0,C 180,E1 -8726.383,E2 -8726.383} C_VEL
LIN {X 0,Y 445.445,Z 476.84,A -85,B 0,C 180,E1 -8727.289,E2 -8727.289} C_VEL
LIN {X 0,Y 445.378,Z 478.245,A -85,B 0,C 180,E1 -8728.193,E2 -8728.193} C_VEL
LIN {X 0,Y 445.368,Z 479.139,A -85,B 0,C 180,E1 -8729.097,E2 -8729.097} C_VEL
LIN {X 0,Y 445.374,Z 479.444,A -85,B 0,C 180,E1 -8730.002,E2 -8730.002} C_VEL
LIN {X 0,Y 445.343,Z 479.17,A -85,B 0,C 180,E1 -8730.906,E2 -8730.906} C_VEL
LIN {X 0,Y 445.379,Z 478.399,A -85,B 0,C 180,E1 -8731.81,E2 -8731.81} C_VEL
LIN {X 0,Y 445.444,Z 477.12,A -85,B 0,C 180,E1 -8732.714,E2 -8732.714} C_VEL
LIN {X 0,Y 445.4,Z 474.097,A -85,B 0,C 180,E1 -8734.073,E2 -8734.073} C_VEL
LIN {X 0,Y 445.515,Z 471.351,A -85,B 0,C 180,E1 -8734.979,E2 -8734.979} C_VEL
LIN {X 0,Y 445.588,Z 465.955,A -85,B 0,C 180,E1 -8736.34,E2 -8736.34} C_VEL
LIN {X 0,Y 445.853,Z 458.836,A -85,B 0,C 180,E1 -8737.701,E2 -8737.701} C_VEL
LIN {X 0,Y 446.124,Z 451.08,A -85,B 0,C 180,E1 -8738.837,E2 -8738.837} C_VEL
LIN {X 0,Y 446.422,Z 444.477,A -85,B 0,C 180,E1 -8739.63,E2 -8739.63} C_VEL
LIN {X 0,Y 446.782,Z 436.501,A -85,B 0,C 180,E1 -8740.423,E2 -8740.423} C_VEL
LIN {X 0,Y 447.109,Z 428.124,A -85,B 0,C 180,E1 -8741.103,E2 -8741.103} C_VEL
LIN {X 0,Y 447.534,Z 417.602,A -85,B 0,C 180,E1 -8741.781,E2 -8741.781} C_VEL
LIN {X 0,Y 447.874,Z 406.567,A -85,B 0,C 180,E1 -8742.289,E2 -8742.289} C_VEL
LIN {X 0,Y 448.162,Z 396.822,A -85,B 0,C 180,E1 -8742.597,E2 -8742.597} C_VEL
LIN {X 0,Y 448.922,Z 336.434,A -85,B 0,C 180,E1 -8743.804,E2 -8743.804} C_VEL
LIN {X 0,Y 446.685,Z 319.434,A -85,B 0,C 180,E1 -8744.25,E2 -8744.25} C_VEL
LIN {X 0,Y 446.377,Z 317.231,A -85,B 0,C 180,E1 -8744.336,E2 -8744.336} C_VEL
LIN {X 0,Y 446.792,Z 299.55,A -85,B 0,C 180,E1 -8747.627,E2 -8747.627} C_VEL
LIN {X 0,Y 447.249,Z 281.535,A -85,B 0,C 180,E1 -8750.947,E2 -8750.947} C_VEL
LIN {X 0,Y 447.21,Z 273.772,A -85,B 0,C 180,E1 -8752.403,E2 -8752.403} C_VEL
LIN {X 0,Y 446.518,Z 269.682,A -85,B 0,C 180,E1 -8753.204,E2 -8753.204} C_VEL
LIN {X 0,Y 446.413,Z 269.693,A -85,B 0,C 180,E1 -8756.182,E2 -8756.182} C_VEL
LIN {X 0,Y 446.421,Z 269.693,A -85,B 0,C 180,E1 -8759.213,E2 -8759.213} C_VEL
LIN {X 0,Y 446.392,Z 269.693,A -85,B 0,C 180,E1 -8762.365,E2 -8762.365} C_VEL
LIN {X 0,Y 446.377,Z 269.693,A -85,B 0,C 180,E1 -8765.631,E2 -8765.631} C_VEL
LIN {X 0,Y 446.4,Z 269.694,A -85,B 0,C 180,E1 -8769.033,E2 -8769.033} C_VEL
LIN {X 0,Y 446.392,Z 269.69,A -85,B 0,C 180,E1 -8772.268,E2 -8772.268} C_VEL
LIN {X 0,Y 446.423,Z 269.69,A -85,B 0,C 180,E1 -8775.109,E2 -8775.109} C_VEL
LIN {X 0,Y 446.415,Z 269.688,A -85,B 0,C 180,E1 -8778.604,E2 -8778.604} C_VEL
LIN {X 0,Y 446.419,Z 269.684,A -85,B 0,C 180,E1 -8781.922,E2 -8781.922} C_VEL
LIN {X 0,Y 446.437,Z 269.686,A -85,B 0,C 180,E1 -8785.474,E2 -8785.474} C_VEL
LIN {X 0,Y 446.43,Z 269.689,A -85,B 0,C 180,E1 -8788.697,E2 -8788.697} C_VEL
LIN {X 0,Y 446.463,Z 269.683,A -85,B 0,C 180,E1 -8791.828,E2 -8791.828} C_VEL
LIN {X 0,Y 446.453,Z 269.691,A -85,B 0,C 180,E1 -8794.844,E2 -8794.844} C_VEL
LIN {X 0,Y 446.463,Z 269.685,A -85,B 0,C 180,E1 -8798.242,E2 -8798.242} C_VEL
LIN {X 0,Y 446.484,Z 269.685,A -85,B 0,C 180,E1 -8801.647,E2 -8801.647} C_VEL
LIN {X 0,Y 446.614,Z 269.743,A -85,B 0,C 180,E1 -8803.336,E2 -8803.336} C_VEL
LIN {X 0,Y 447.265,Z 273.685,A -85,B 0,C 180,E1 -8803.949,E2 -8803.949} C_VEL
LIN {X 0,Y 446.967,Z 285.705,A -85,B 0,C 180,E1 -8805.719,E2 -8805.719} C_VEL
LIN {X 0,Y 449.352,Z 301.036,A -85,B 0,C 180,E1 -8806.151,E2 -8806.151} C_VEL
LIN {X 0,Y 448.367,Z 366.25,A -85,B 0,C 180,E1 -8807.463,E2 -8807.463} C_VEL
LIN {X 0,Y 448.054,Z 378.532,A -85,B 0,C 180,E1 -8807.886,E2 -8807.886} C_VEL
LIN {X 0,Y 447.787,Z 387.448,A -85,B 0,C 180,E1 -8808.338,E2 -8808.338} C_VEL
LIN {X 0,Y 447.454,Z 397.59,A -85,B 0,C 180,E1 -8809.017,E2 -8809.017} C_VEL
LIN {X 0,Y 447.205,Z 405.643,A -85,B 0,C 180,E1 -8809.698,E2 -8809.698} C_VEL
LIN {X 0,Y 446.922,Z 413.333,A -85,B 0,C 180,E1 -8810.492,E2 -8810.492} C_VEL
LIN {X 0,Y 446.473,Z 422.227,A -85,B 0,C 180,E1 -8811.624,E2 -8811.624} C_VEL
LIN {X 0,Y 446.164,Z 429.078,A -85,B 0,C 180,E1 -8812.756,E2 -8812.756} C_VEL
LIN {X 0,Y 446.074,Z 433.579,A -85,B 0,C 180,E1 -8813.664,E2 -8813.664} C_VEL
LIN {X 0,Y 445.716,Z 437.333,A -85,B 0,C 180,E1 -8814.567,E2 -8814.567} C_VEL
LIN {X 0,Y 445.746,Z 440.368,A -85,B 0,C 180,E1 -8815.474,E2 -8815.474} C_VEL
LIN {X 0,Y 445.662,Z 442.724,A -85,B 0,C 180,E1 -8816.379,E2 -8816.379} C_VEL
LIN {X 0,Y 445.521,Z 444.487,A -85,B 0,C 180,E1 -8817.283,E2 -8817.283} C_VEL
LIN {X 0,Y 445.435,Z 445.725,A -85,B 0,C 180,E1 -8818.187,E2 -8818.187} C_VEL
LIN {X 0,Y 445.373,Z 446.461,A -85,B 0,C 180,E1 -8819.091,E2 -8819.091} C_VEL
LIN {X 0,Y 445.376,Z 446.694,A -85,B 0,C 180,E1 -8819.995,E2 -8819.995} C_VEL
LIN {X 0,Y 445.372,Z 446.332,A -85,B 0,C 180,E1 -8820.9,E2 -8820.9} C_VEL
LIN {X 0,Y 445.408,Z 445.418,A -85,B 0,C 180,E1 -8821.804,E2 -8821.804} C_VEL
LIN {X 0,Y 445.501,Z 443.994,A -85,B 0,C 180,E1 -8822.708,E2 -8822.708} C_VEL
LIN {X 0,Y 445.637,Z 440.84,A -85,B 0,C 180,E1 -8824.065,E2 -8824.065} C_VEL
LIN {X 0,Y 445.683,Z 436.331,A -85,B 0,C 180,E1 -8825.424,E2 -8825.424} C_VEL
LIN {X 0,Y 445.988,Z 430.911,A -85,B 0,C 180,E1 -8826.625,E2 -8826.625} C_VEL
LIN {X 0,Y 446.101,Z 424.887,A -85,B 0,C 180,E1 -8827.691,E2 -8827.691} C_VEL
LIN {X 0,Y 446.326,Z 418.623,A -85,B 0,C 180,E1 -8828.598,E2 -8828.598} C_VEL
LIN {X 0,Y 446.578,Z 412.045,A -85,B 0,C 180,E1 -8829.392,E2 -8829.392} C_VEL
LIN {X 0,Y 446.89,Z 404.094,A -85,B 0,C 180,E1 -8830.185,E2 -8830.185} C_VEL
LIN {X 0,Y 447.117,Z 395.711,A -85,B 0,C 180,E1 -8830.867,E2 -8830.867} C_VEL
LIN {X 0,Y 447.461,Z 385.063,A -85,B 0,C 180,E1 -8831.547,E2 -8831.547} C_VEL
LIN {X 0,Y 447.721,Z 373.657,A -85,B 0,C 180,E1 -8832.057,E2 -8832.057} C_VEL
LIN {X 0,Y 447.869,Z 364.5,A -85,B 0,C 180,E1 -8832.34,E2 -8832.34} C_VEL
LIN {X 0,Y 448.454,Z 300.664,A -85,B 0,C 180,E1 -8833.556,E2 -8833.556} C_VEL
LIN {X 0,Y 446.413,Z 287.673,A -85,B 0,C 180,E1 -8833.886,E2 -8833.886} C_VEL
LIN {X 0,Y 446.718,Z 275.981,A -85,B 0,C 180,E1 -8836.915,E2 -8836.915} C_VEL
LIN {X 0,Y 446.537,Z 269.678,A -85,B 0,C 180,E1 -8838.618,E2 -8838.618} C_VEL
LIN {X 0,Y 446.404,Z 269.69,A -85,B 0,C 180,E1 -8842.194,E2 -8842.194} C_VEL
LIN {X 0,Y 446.415,Z 269.69,A -85,B 0,C 180,E1 -8845.148,E2 -8845.148} C_VEL
LIN {X 0,Y 446.399,Z 269.691,A -85,B 0,C 180,E1 -8848.178,E2 -8848.178} C_VEL
LIN {X 0,Y 446.389,Z 269.693,A -85,B 0,C 180,E1 -8851.295,E2 -8851.295} C_VEL
LIN {X 0,Y 446.404,Z 269.69,A -85,B 0,C 180,E1 -8854.517,E2 -8854.517} C_VEL
LIN {X 0,Y 446.383,Z 269.694,A -85,B 0,C 180,E1 -8858.073,E2 -8858.073} C_VEL
LIN {X 0,Y 446.388,Z 269.694,A -85,B 0,C 180,E1 -8861.387,E2 -8861.387} C_VEL
LIN {X 0,Y 446.417,Z 269.69,A -85,B 0,C 180,E1 -8865.098,E2 -8865.098} C_VEL
LIN {X 0,Y 446.392,Z 269.692,A -85,B 0,C 180,E1 -8868.604,E2 -8868.604} C_VEL
LIN {X 0,Y 446.374,Z 269.695,A -85,B 0,C 180,E1 -8871.916,E2 -8871.916} C_VEL
LIN {X 0,Y 446.388,Z 269.694,A -85,B 0,C 180,E1 -8875.472,E2 -8875.472} C_VEL
LIN {X 0,Y 446.371,Z 269.695,A -85,B 0,C 180,E1 -8878.695,E2 -8878.695} C_VEL
LIN {X 0,Y 446.439,Z 269.689,A -85,B 0,C 180,E1 -8881.817,E2 -8881.817} C_VEL
LIN {X 0,Y 446.409,Z 269.69,A -85,B 0,C 180,E1 -8884.844,E2 -8884.844} C_VEL
LIN {X 0,Y 446.397,Z 269.693,A -85,B 0,C 180,E1 -8888.241,E2 -8888.241} C_VEL
LIN {X 0,Y 446.403,Z 269.691,A -85,B 0,C 180,E1 -8891.646,E2 -8891.646} C_VEL
LIN {X 0,Y 446.443,Z 269.686,A -85,B 0,C 180,E1 -8894.287,E2 -8894.287} C_VEL
LIN {X 0,Y 445.814,Z 269.766,A -85,B 0,C 180,E1 -8895.04,E2 -8895.04} C_VEL
LIN {X 0,Y 443.006,Z 270.118,A -85,B 0,C 180,E1 -8896.263,E2 -8896.263} C_VEL
LIN {X 0,Y 440.594,Z 270.417,A -85,B 0,C 180,E1 -8897.25,E2 -8897.25} C_VEL
LIN {X 0,Y 439.53,Z 270.548,A -85,B 0,C 180,E1 -8898.012,E2 -8898.012} C_VEL
LIN {X 0,Y 439.429,Z 270.559,A -85,B 0,C 180,E1 -8898.27,E2 -8898.27} C_VEL
LIN {X 0,Y 439.491,Z 270.551,A -85,B 0,C 180,E1 -8901.724,E2 -8901.724} C_VEL
LIN {X 0,Y 439.568,Z 270.544,A -85,B 0,C 180,E1 -8904.494,E2 -8904.494} C_VEL
LIN {X 0,Y 439.579,Z 270.541,A -85,B 0,C 180,E1 -8908.166,E2 -8908.166} C_VEL
LIN {X 0,Y 439.704,Z 270.525,A -85,B 0,C 180,E1 -8909.998,E2 -8909.998} C_VEL
LIN {X 0,Y 439.605,Z 270.539,A -85,B 0,C 180,E1 -8912.747,E2 -8912.747} C_VEL
LIN {X 0,Y 439.561,Z 270.544,A -85,B 0,C 180,E1 -8916.424,E2 -8916.424} C_VEL
LIN {X 0,Y 439.446,Z 270.558,A -85,B 0,C 180,E1 -8919.201,E2 -8919.201} C_VEL
LIN {X 0,Y 439.444,Z 270.559,A -85,B 0,C 180,E1 -8922.727,E2 -8922.727} C_VEL
LIN {X 0,Y 439.387,Z 270.564,A -85,B 0,C 180,E1 -8926.349,E2 -8926.349} C_VEL
LIN {X 0,Y 439.343,Z 270.571,A -85,B 0,C 180,E1 -8929.627,E2 -8929.627} C_VEL
LIN {X 0,Y 439.307,Z 270.574,A -85,B 0,C 180,E1 -8932.577,E2 -8932.577} C_VEL
LIN {X 0,Y 439.355,Z 270.569,A -85,B 0,C 180,E1 -8935.586,E2 -8935.586} C_VEL
LIN {X 0,Y 439.368,Z 270.567,A -85,B 0,C 180,E1 -8938.675,E2 -8938.675} C_VEL
LIN {X 0,Y 439.318,Z 270.574,A -85,B 0,C 180,E1 -8941.863,E2 -8941.863} C_VEL
LIN {X 0,Y 439.346,Z 270.57,A -85,B 0,C 180,E1 -8945.158,E2 -8945.158} C_VEL
LIN {X 0,Y 439.349,Z 270.57,A -85,B 0,C 180,E1 -8948.596,E2 -8948.596} C_VEL
LIN {X 0,Y 439.354,Z 270.569,A -85,B 0,C 180,E1 -8951.262,E2 -8951.262} C_VEL
LIN {X 0,Y 439.36,Z 270.569,A -85,B 0,C 180,E1 -8954.731,E2 -8954.731} C_VEL
LIN {X 0,Y 439.365,Z 270.57,A -85,B 0,C 180,E1 -8957.801,E2 -8957.801} C_VEL
LIN {X 0,Y 439.405,Z 270.563,A -85,B 0,C 180,E1 -8960.234,E2 -8960.234} C_VEL
LIN {X 0,Y 439.334,Z 270.572,A -85,B 0,C 180,E1 -8963.717,E2 -8963.717} C_VEL
LIN {X 0,Y 439.331,Z 270.572,A -85,B 0,C 180,E1 -8967.058,E2 -8967.058} C_VEL
LIN {X 0,Y 439.342,Z 270.572,A -85,B 0,C 180,E1 -8970.278,E2 -8970.278} C_VEL
LIN {X 0,Y 439.382,Z 270.565,A -85,B 0,C 180,E1 -8973.4,E2 -8973.4} C_VEL
LIN {X 0,Y 439.348,Z 270.572,A -85,B 0,C 180,E1 -8976.434,E2 -8976.434} C_VEL
LIN {X 0,Y 439.355,Z 270.569,A -85,B 0,C 180,E1 -8979.402,E2 -8979.402} C_VEL
LIN {X 0,Y 439.374,Z 270.568,A -85,B 0,C 180,E1 -8982.313,E2 -8982.313} C_VEL
LIN {X 0,Y 439.418,Z 270.561,A -85,B 0,C 180,E1 -8985.179,E2 -8985.179} C_VEL
LIN {X 0,Y 439.457,Z 270.555,A -85,B 0,C 180,E1 -8988.006,E2 -8988.006} C_VEL
LIN {X 0,Y 439.48,Z 270.554,A -85,B 0,C 180,E1 -8991.73,E2 -8991.73} C_VEL
LIN {X 0,Y 439.589,Z 270.54,A -85,B 0,C 180,E1 -8994.5,E2 -8994.5} C_VEL
LIN {X 0,Y 439.608,Z 270.537,A -85,B 0,C 180,E1 -8998.172,E2 -8998.172} C_VEL
LIN {X 0,Y 439.671,Z 270.53,A -85,B 0,C 180,E1 -9000.005,E2 -9000.005} C_VEL
LIN {X 0,Y 439.613,Z 270.537,A -85,B 0,C 180,E1 -9002.753,E2 -9002.753} C_VEL
LIN {X 0,Y 439.549,Z 270.544,A -85,B 0,C 180,E1 -9006.43,E2 -9006.43} C_VEL
LIN {X 0,Y 439.481,Z 270.556,A -85,B 0,C 180,E1 -9009.206,E2 -9009.206} C_VEL
LIN {X 0,Y 439.454,Z 270.556,A -85,B 0,C 180,E1 -9012.942,E2 -9012.942} C_VEL
LIN {X 0,Y 439.392,Z 270.565,A -85,B 0,C 180,E1 -9016.332,E2 -9016.332} C_VEL
LIN {X 0,Y 439.393,Z 270.566,A -85,B 0,C 180,E1 -9019.63,E2 -9019.63} C_VEL
LIN {X 0,Y 439.355,Z 270.569,A -85,B 0,C 180,E1 -9022.58,E2 -9022.58} C_VEL
LIN {X 0,Y 439.36,Z 270.57,A -85,B 0,C 180,E1 -9025.591,E2 -9025.591} C_VEL
LIN {X 0,Y 439.392,Z 270.565,A -85,B 0,C 180,E1 -9028.679,E2 -9028.679} C_VEL
LIN {X 0,Y 439.362,Z 270.569,A -85,B 0,C 180,E1 -9032.033,E2 -9032.033} C_VEL
LIN {X 0,Y 439.385,Z 270.564,A -85,B 0,C 180,E1 -9035.342,E2 -9035.342} C_VEL
LIN {X 0,Y 439.352,Z 270.569,A -85,B 0,C 180,E1 -9038.601,E2 -9038.601} C_VEL
LIN {X 0,Y 439.349,Z 270.572,A -85,B 0,C 180,E1 -9042.213,E2 -9042.213} C_VEL
LIN {X 0,Y 439.371,Z 270.567,A -85,B 0,C 180,E1 -9045.27,E2 -9045.27} C_VEL
LIN {X 0,Y 439.353,Z 270.57,A -85,B 0,C 180,E1 -9049.019,E2 -9049.019} C_VEL
LIN {X 0,Y 439.343,Z 270.572,A -85,B 0,C 180,E1 -9052.567,E2 -9052.567} C_VEL
LIN {X 0,Y 439.395,Z 270.564,A -85,B 0,C 180,E1 -9054.846,E2 -9054.846} C_VEL
LIN {X 0,Y 439.368,Z 270.567,A -85,B 0,C 180,E1 -9058.141,E2 -9058.141} C_VEL
LIN {X 0,Y 439.39,Z 270.565,A -85,B 0,C 180,E1 -9061.612,E2 -9061.612} C_VEL
LIN {X 0,Y 439.467,Z 270.742,A -85,B 0,C 180,E1 -9065.37,E2 -9065.37} C_VEL
LIN {X 0,Y 440.931,Z 280.115,A -85,B 0,C 180,E1 -9067.511,E2 -9067.511} C_VEL
LIN {X 0,Y 440.482,Z 291.523,A -85,B 0,C 180,E1 -9069.989,E2 -9069.989} C_VEL
LIN {X 0,Y 439.716,Z 308.082,A -85,B 0,C 180,E1 -9073.538,E2 -9073.538} C_VEL
LIN {X 0,Y 439.308,Z 319.407,A -85,B 0,C 180,E1 -9075.94,E2 -9075.94} C_VEL
LIN {X 0,Y 441.448,Z 339.096,A -85,B 0,C 180,E1 -9076.401,E2 -9076.401} C_VEL
LIN {X 0,Y 440.79,Z 397.441,A -85,B 0,C 180,E1 -9077.543,E2 -9077.543} C_VEL
LIN {X 0,Y 440.467,Z 408.821,A -85,B 0,C 180,E1 -9077.913,E2 -9077.913} C_VEL
LIN {X 0,Y 440.109,Z 420.19,A -85,B 0,C 180,E1 -9078.488,E2 -9078.488} C_VEL
LIN {X 0,Y 439.778,Z 428.81,A -85,B 0,C 180,E1 -9079.062,E2 -9079.062} C_VEL
LIN {X 0,Y 439.552,Z 437.127,A -85,B 0,C 180,E1 -9079.756,E2 -9079.756} C_VEL
LIN {X 0,Y 439.196,Z 445.018,A -85,B 0,C 180,E1 -9080.561,E2 -9080.561} C_VEL
LIN {X 0,Y 438.918,Z 452.427,A -85,B 0,C 180,E1 -9081.484,E2 -9081.484} C_VEL
LIN {X 0,Y 438.683,Z 459.919,A -85,B 0,C 180,E1 -9082.638,E2 -9082.638} C_VEL
LIN {X 0,Y 438.452,Z 466.232,A -85,B 0,C 180,E1 -9083.906,E2 -9083.906} C_VEL
LIN {X 0,Y 438.443,Z 470.352,A -85,B 0,C 180,E1 -9084.944,E2 -9084.944} C_VEL
LIN {X 0,Y 438.322,Z 474.484,A -85,B 0,C 180,E1 -9086.324,E2 -9086.324} C_VEL
LIN {X 0,Y 438.372,Z 476.479,A -85,B 0,C 180,E1 -9087.245,E2 -9087.245} C_VEL
LIN {X 0,Y 438.299,Z 477.924,A -85,B 0,C 180,E1 -9088.164,E2 -9088.164} C_VEL
LIN {X 0,Y 438.28,Z 478.845,A -85,B 0,C 180,E1 -9089.083,E2 -9089.083} C_VEL
LIN {X 0,Y 438.284,Z 479.157,A -85,B 0,C 180,E1 -9090.002,E2 -9090.002} C_VEL
LIN {X 0,Y 438.257,Z 478.913,A -85,B 0,C 180,E1 -9090.92,E2 -9090.92} C_VEL
LIN {X 0,Y 438.3,Z 478.17,A -85,B 0,C 180,E1 -9091.839,E2 -9091.839} C_VEL
LIN {X 0,Y 438.353,Z 476.913,A -85,B 0,C 180,E1 -9092.758,E2 -9092.758} C_VEL
LIN {X 0,Y 438.314,Z 473.904,A -85,B 0,C 180,E1 -9094.139,E2 -9094.139} C_VEL
LIN {X 0,Y 438.447,Z 471.178,A -85,B 0,C 180,E1 -9095.059,E2 -9095.059} C_VEL
LIN {X 0,Y 438.469,Z 467.228,A -85,B 0,C 180,E1 -9096.112,E2 -9096.112} C_VEL
LIN {X 0,Y 438.658,Z 462.456,A -85,B 0,C 180,E1 -9097.134,E2 -9097.134} C_VEL
LIN {X 0,Y 438.842,Z 457.245,A -85,B 0,C 180,E1 -9098.057,E2 -9098.057} C_VEL
LIN {X 0,Y 439.105,Z 451.001,A -85,B 0,C 180,E1 -9098.979,E2 -9098.979} C_VEL
LIN {X 0,Y 439.499,Z 443.424,A -85,B 0,C 180,E1 -9099.9,E2 -9099.9} C_VEL
LIN {X 0,Y 439.854,Z 435.335,A -85,B 0,C 180,E1 -9100.706,E2 -9100.706} C_VEL
LIN {X 0,Y 440.268,Z 425.285,A -85,B 0,C 180,E1 -9101.511,E2 -9101.511} C_VEL
LIN {X 0,Y 440.741,Z 414.692,A -85,B 0,C 180,E1 -9102.141,E2 -9102.141} C_VEL
LIN {X 0,Y 441.03,Z 405.766,A -85,B 0,C 180,E1 -9102.541,E2 -9102.541} C_VEL
LIN {X 0,Y 441.337,Z 395.825,A -85,B 0,C 180,E1 -9102.854,E2 -9102.854} C_VEL
LIN {X 0,Y 442.095,Z 336.727,A -85,B 0,C 180,E1 -9104.066,E2 -9104.066} C_VEL
LIN {X 0,Y 440.015,Z 320.691,A -85,B 0,C 180,E1 -9104.511,E2 -9104.511} C_VEL
LIN {X 0,Y 439.394,Z 316.931,A -85,B 0,C 180,E1 -9104.642,E2 -9104.642} C_VEL
LIN {X 0,Y 439.824,Z 300.78,A -85,B 0,C 180,E1 -9107.676,E2 -9107.676} C_VEL
LIN {X 0,Y 440.295,Z 282.772,A -85,B 0,C 180,E1 -9111.049,E2 -9111.049} C_VEL
LIN {X 0,Y 440.227,Z 274.881,A -85,B 0,C 180,E1 -9112.53,E2 -9112.53} C_VEL
LIN {X 0,Y 439.462,Z 270.559,A -85,B 0,C 180,E1 -9113.411,E2 -9113.411} C_VEL
LIN {X 0,Y 439.361,Z 270.574,A -85,B 0,C 180,E1 -9116.61,E2 -9116.61} C_VEL
LIN {X 0,Y 439.37,Z 270.569,A -85,B 0,C 180,E1 -9119.728,E2 -9119.728} C_VEL
LIN {X 0,Y 439.332,Z 270.575,A -85,B 0,C 180,E1 -9122.951,E2 -9122.951} C_VEL
LIN {X 0,Y 439.355,Z 270.569,A -85,B 0,C 180,E1 -9126.29,E2 -9126.29} C_VEL
LIN {X 0,Y 439.361,Z 270.568,A -85,B 0,C 180,E1 -9128.599,E2 -9128.599} C_VEL
LIN {X 0,Y 439.359,Z 270.565,A -85,B 0,C 180,E1 -9132.21,E2 -9132.21} C_VEL
LIN {X 0,Y 439.379,Z 270.566,A -85,B 0,C 180,E1 -9135.265,E2 -9135.265} C_VEL
LIN {X 0,Y 439.378,Z 270.566,A -85,B 0,C 180,E1 -9138.746,E2 -9138.746} C_VEL
LIN {X 0,Y 439.375,Z 270.562,A -85,B 0,C 180,E1 -9141.609,E2 -9141.609} C_VEL
LIN {X 0,Y 439.41,Z 270.563,A -85,B 0,C 180,E1 -9144.842,E2 -9144.842} C_VEL
LIN {X 0,Y 439.385,Z 270.564,A -85,B 0,C 180,E1 -9148.137,E2 -9148.137} C_VEL
LIN {X 0,Y 439.417,Z 270.563,A -85,B 0,C 180,E1 -9151.604,E2 -9151.604} C_VEL
LIN {X 0,Y 439.391,Z 270.567,A -85,B 0,C 180,E1 -9154.411,E2 -9154.411} C_VEL
LIN {X 0,Y 439.378,Z 270.571,A -85,B 0,C 180,E1 -9157.422,E2 -9157.422} C_VEL
LIN {X 0,Y 439.455,Z 270.559,A -85,B 0,C 180,E1 -9160.66,E2 -9160.66} C_VEL
LIN {X 0,Y 439.559,Z 270.711,A -85,B 0,C 180,E1 -9163.091,E2 -9163.091} C_VEL
LIN {X 0,Y 440.376,Z 274.177,A -85,B 0,C 180,E1 -9163.647,E2 -9163.647} C_VEL
LIN {X 0,Y 440.121,Z 285.959,A -85,B 0,C 180,E1 -9165.406,E2 -9165.406} C_VEL
LIN {X 0,Y 442.555,Z 301.139,A -85,B 0,C 180,E1 -9165.862,E2 -9165.862} C_VEL
LIN {X 0,Y 441.509,Z 366.984,A -85,B 0,C 180,E1 -9167.236,E2 -9167.236} C_VEL
LIN {X 0,Y 441.169,Z 379.625,A -85,B 0,C 180,E1 -9167.694,E2 -9167.694} C_VEL
LIN {X 0,Y 440.889,Z 388.364,A -85,B 0,C 180,E1 -9168.153,E2 -9168.153} C_VEL
LIN {X 0,Y 440.625,Z 396.904,A -85,B 0,C 180,E1 -9168.729,E2 -9168.729} C_VEL
LIN {X 0,Y 440.291,Z 405.138,A -85,B 0,C 180,E1 -9169.418,E2 -9169.418} C_VEL
LIN {X 0,Y 440.001,Z 412.966,A -85,B 0,C 180,E1 -9170.225,E2 -9170.225} C_VEL
LIN {X 0,Y 439.659,Z 419.45,A -85,B 0,C 180,E1 -9171.029,E2 -9171.029} C_VEL
LIN {X 0,Y 439.306,Z 425.624,A -85,B 0,C 180,E1 -9171.949,E2 -9171.949} C_VEL
LIN {X 0,Y 439.145,Z 430.687,A -85,B 0,C 180,E1 -9172.862,E2 -9172.862} C_VEL
LIN {X 0,Y 438.849,Z 435.952,A -85,B 0,C 180,E1 -9174.021,E2 -9174.021} C_VEL
LIN {X 0,Y 438.681,Z 440.744,A -85,B 0,C 180,E1 -9175.401,E2 -9175.401} C_VEL
LIN {X 0,Y 438.606,Z 443.093,A -85,B 0,C 180,E1 -9176.321,E2 -9176.321} C_VEL
LIN {X 0,Y 438.453,Z 444.833,A -85,B 0,C 180,E1 -9177.239,E2 -9177.239} C_VEL
LIN {X 0,Y 438.354,Z 446.045,A -85,B 0,C 180,E1 -9178.158,E2 -9178.158} C_VEL
LIN {X 0,Y 438.286,Z 446.751,A -85,B 0,C 180,E1 -9179.077,E2 -9179.077} C_VEL
LIN {X 0,Y 438.286,Z 446.956,A -85,B 0,C 180,E1 -9179.995,E2 -9179.995} C_VEL
LIN {X 0,Y 438.284,Z 446.583,A -85,B 0,C 180,E1 -9180.914,E2 -9180.914} C_VEL
LIN {X 0,Y 438.328,Z 445.63,A -85,B 0,C 180,E1 -9181.833,E2 -9181.833} C_VEL
LIN {X 0,Y 438.468,Z 443.303,A -85,B 0,C 180,E1 -9183.211,E2 -9183.211} C_VEL
LIN {X 0,Y 438.492,Z 439.59,A -85,B 0,C 180,E1 -9184.592,E2 -9184.592} C_VEL
LIN {X 0,Y 438.61,Z 436.366,A -85,B 0,C 180,E1 -9185.512,E2 -9185.512} C_VEL
LIN {X 0,Y 438.883,Z 431.515,A -85,B 0,C 180,E1 -9186.608,E2 -9186.608} C_VEL
LIN {X 0,Y 439.012,Z 426.215,A -85,B 0,C 180,E1 -9187.584,E2 -9187.584} C_VEL
LIN {X 0,Y 439.217,Z 420.149,A -85,B 0,C 180,E1 -9188.507,E2 -9188.507} C_VEL
LIN {X 0,Y 439.506,Z 412.769,A -85,B 0,C 180,E1 -9189.428,E2 -9189.428} C_VEL
LIN {X 0,Y 439.832,Z 404.902,A -85,B 0,C 180,E1 -9190.234,E2 -9190.234} C_VEL
LIN {X 0,Y 440.074,Z 396.632,A -85,B 0,C 180,E1 -9190.927,E2 -9190.927} C_VEL
LIN {X 0,Y 440.433,Z 386.197,A -85,B 0,C 180,E1 -9191.617,E2 -9191.617} C_VEL
LIN {X 0,Y 440.724,Z 374.548,A -85,B 0,C 180,E1 -9192.163,E2 -9192.163} C_VEL
LIN {X 0,Y 440.855,Z 364.531,A -85,B 0,C 180,E1 -9192.481,E2 -9192.481} C_VEL
LIN {X 0,Y 441.422,Z 301.098,A -85,B 0,C 180,E1 -9193.725,E2 -9193.725} C_VEL
LIN {X 0,Y 439.364,Z 287.945,A -85,B 0,C 180,E1 -9194.054,E2 -9194.054} C_VEL
LIN {X 0,Y 439.707,Z 275.99,A -85,B 0,C 180,E1 -9197.193,E2 -9197.193} C_VEL
LIN {X 0,Y 439.489,Z 270.555,A -85,B 0,C 180,E1 -9198.692,E2 -9198.692} C_VEL
LIN {X 0,Y 439.376,Z 270.566,A -85,B 0,C 180,E1 -9201.914,E2 -9201.914} C_VEL
LIN {X 0,Y 439.375,Z 270.568,A -85,B 0,C 180,E1 -9204.568,E2 -9204.568} C_VEL
LIN {X 0,Y 439.33,Z 270.574,A -85,B 0,C 180,E1 -9207.633,E2 -9207.633} C_VEL
LIN {X 0,Y 439.335,Z 270.573,A -85,B 0,C 180,E1 -9210.783,E2 -9210.783} C_VEL
LIN {X 0,Y 439.364,Z 270.568,A -85,B 0,C 180,E1 -9214.038,E2 -9214.038} C_VEL
LIN {X 0,Y 439.32,Z 270.574,A -85,B 0,C 180,E1 -9216.881,E2 -9216.881} C_VEL
LIN {X 0,Y 439.348,Z 270.571,A -85,B 0,C 180,E1 -9219.839,E2 -9219.839} C_VEL
LIN {X 0,Y 439.339,Z 270.57,A -85,B 0,C 180,E1 -9222.619,E2 -9222.619} C_VEL
LIN {X 0,Y 439.365,Z 270.57,A -85,B 0,C 180,E1 -9225.265,E2 -9225.265} C_VEL
LIN {X 0,Y 439.352,Z 270.569,A -85,B 0,C 180,E1 -9228.738,E2 -9228.738} C_VEL
LIN {X 0,Y 439.33,Z 270.573,A -85,B 0,C 180,E1 -9231.603,E2 -9231.603} C_VEL
LIN {X 0,Y 439.359,Z 270.568,A -85,B 0,C 180,E1 -9234.839,E2 -9234.839} C_VEL
LIN {X 0,Y 439.328,Z 270.573,A -85,B 0,C 180,E1 -9238.135,E2 -9238.135} C_VEL
LIN {X 0,Y 439.386,Z 270.566,A -85,B 0,C 180,E1 -9241.594,E2 -9241.594} C_VEL
LIN {X 0,Y 439.357,Z 270.569,A -85,B 0,C 180,E1 -9244.411,E2 -9244.411} C_VEL
LIN {X 0,Y 439.314,Z 270.573,A -85,B 0,C 180,E1 -9247.42,E2 -9247.42} C_VEL
LIN {X 0,Y 439.389,Z 270.565,A -85,B 0,C 180,E1 -9250.659,E2 -9250.659} C_VEL
LIN {X 0,Y 439.403,Z 270.564,A -85,B 0,C 180,E1 -9254.279,E2 -9254.279} C_VEL
LIN {X 0,Y 439.457,Z 270.557,A -85,B 0,C 180,E1 -9257.999,E2 -9257.999} C_VEL
LIN {X 0,Y 439.429,Z 270.559,A -85,B 0,C 180,E1 -9258.27,E2 -9258.27} C_VEL
LIN {X 0,Y 438.754,Z 270.645,A -85,B 0,C 180,E1 -9259.035,E2 -9259.035} C_VEL
LIN {X 0,Y 436.006,Z 270.99,A -85,B 0,C 180,E1 -9260.279,E2 -9260.279} C_VEL
LIN {X 0,Y 433.674,Z 271.283,A -85,B 0,C 180,E1 -9261.283,E2 -9261.283} C_VEL
LIN {X 0,Y 432.636,Z 271.41,A -85,B 0,C 180,E1 -9262.057,E2 -9262.057} C_VEL
LIN {X 0,Y 432.529,Z 271.421,A -85,B 0,C 180,E1 -9262.319,E2 -9262.319} C_VEL
LIN {X 0,Y 432.544,Z 271.419,A -85,B 0,C 180,E1 -9264.404,E2 -9264.404} C_VEL
LIN {X 0,Y 432.549,Z 271.417,A -85,B 0,C 180,E1 -9268.136,E2 -9268.136} C_VEL
LIN {X 0,Y 432.675,Z 271.401,A -85,B 0,C 180,E1 -9269.998,E2 -9269.998} C_VEL
LIN {X 0,Y 432.555,Z 271.417,A -85,B 0,C 180,E1 -9272.792,E2 -9272.792} C_VEL
LIN {X 0,Y 432.515,Z 271.422,A -85,B 0,C 180,E1 -9276.53,E2 -9276.53} C_VEL
LIN {X 0,Y 432.389,Z 271.437,A -85,B 0,C 180,E1 -9279.353,E2 -9279.353} C_VEL
LIN {X 0,Y 432.385,Z 271.44,A -85,B 0,C 180,E1 -9282.812,E2 -9282.812} C_VEL
LIN {X 0,Y 432.352,Z 271.441,A -85,B 0,C 180,E1 -9286.479,E2 -9286.479} C_VEL
LIN {X 0,Y 432.279,Z 271.452,A -85,B 0,C 180,E1 -9289.961,E2 -9289.961} C_VEL
LIN {X 0,Y 432.261,Z 271.454,A -85,B 0,C 180,E1 -9292.965,E2 -9292.965} C_VEL
LIN {X 0,Y 432.31,Z 271.447,A -85,B 0,C 180,E1 -9296.034,E2 -9296.034} C_VEL
LIN {X 0,Y 432.295,Z 271.45,A -85,B 0,C 180,E1 -9299.189,E2 -9299.189} C_VEL
LIN {X 0,Y 432.27,Z 271.453,A -85,B 0,C 180,E1 -9302.295,E2 -9302.295} C_VEL
LIN {X 0,Y 432.286,Z 271.449,A -85,B 0,C 180,E1 -9304.68,E2 -9304.68} C_VEL
LIN {X 0,Y 432.302,Z 271.448,A -85,B 0,C 180,E1 -9308.151,E2 -9308.151} C_VEL
LIN {X 0,Y 432.323,Z 271.448,A -85,B 0,C 180,E1 -9311.611,E2 -9311.611} C_VEL
LIN {X 0,Y 432.33,Z 271.444,A -85,B 0,C 180,E1 -9314.345,E2 -9314.345} C_VEL
LIN {X 0,Y 432.318,Z 271.445,A -85,B 0,C 180,E1 -9317.013,E2 -9317.013} C_VEL
LIN {X 0,Y 432.312,Z 271.449,A -85,B 0,C 180,E1 -9319.821,E2 -9319.821} C_VEL
LIN {X 0,Y 432.273,Z 271.451,A -85,B 0,C 180,E1 -9323.027,E2 -9323.027} C_VEL
LIN {X 0,Y 432.318,Z 271.448,A -85,B 0,C 180,E1 -9326.001,E2 -9326.001} C_VEL
LIN {X 0,Y 432.308,Z 271.446,A -85,B 0,C 180,E1 -9329.494,E2 -9329.494} C_VEL
LIN {X 0,Y 432.348,Z 271.442,A -85,B 0,C 180,E1 -9332.932,E2 -9332.932} C_VEL
LIN {X 0,Y 432.331,Z 271.444,A -85,B 0,C 180,E1 -9336.028,E2 -9336.028} C_VEL
LIN {X 0,Y 432.317,Z 271.446,A -85,B 0,C 180,E1 -9339.051,E2 -9339.051} C_VEL
LIN {X 0,Y 432.33,Z 271.444,A -85,B 0,C 180,E1 -9342.015,E2 -9342.015} C_VEL
LIN {X 0,Y 432.366,Z 271.44,A -85,B 0,C 180,E1 -9344.931,E2 -9344.931} C_VEL
LIN {X 0,Y 432.433,Z 271.431,A -85,B 0,C 180,E1 -9347.808,E2 -9347.808} C_VEL
LIN {X 0,Y 432.44,Z 271.431,A -85,B 0,C 180,E1 -9351.595,E2 -9351.595} C_VEL
LIN {X 0,Y 432.565,Z 271.415,A -85,B 0,C 180,E1 -9354.411,E2 -9354.411} C_VEL
LIN {X 0,Y 432.577,Z 271.413,A -85,B 0,C 180,E1 -9358.143,E2 -9358.143} C_VEL
LIN {X 0,Y 432.622,Z 271.408,A -85,B 0,C 180,E1 -9360.005,E2 -9360.005} C_VEL
LIN {X 0,Y 432.565,Z 271.416,A -85,B 0,C 180,E1 -9362.798,E2 -9362.798} C_VEL
LIN {X 0,Y 432.561,Z 271.415,A -85,B 0,C 180,E1 -9365.599,E2 -9365.599} C_VEL
LIN {X 0,Y 432.45,Z 271.429,A -85,B 0,C 180,E1 -9368.415,E2 -9368.415} C_VEL
LIN {X 0,Y 432.448,Z 271.43,A -85,B 0,C 180,E1 -9372.201,E2 -9372.201} C_VEL
LIN {X 0,Y 432.379,Z 271.438,A -85,B 0,C 180,E1 -9376.045,E2 -9376.045} C_VEL
LIN {X 0,Y 432.379,Z 271.441,A -85,B 0,C 180,E1 -9379.489,E2 -9379.489} C_VEL
LIN {X 0,Y 432.303,Z 271.447,A -85,B 0,C 180,E1 -9382.969,E2 -9382.969} C_VEL
LIN {X 0,Y 432.314,Z 271.446,A -85,B 0,C 180,E1 -9386.039,E2 -9386.039} C_VEL
LIN {X 0,Y 432.327,Z 271.444,A -85,B 0,C 180,E1 -9389.192,E2 -9389.192} C_VEL
LIN {X 0,Y 432.318,Z 271.445,A -85,B 0,C 180,E1 -9392.447,E2 -9392.447} C_VEL
LIN {X 0,Y 432.331,Z 271.446,A -85,B 0,C 180,E1 -9395.822,E2 -9395.822} C_VEL
LIN {X 0,Y 432.298,Z 271.447,A -85,B 0,C 180,E1 -9399.352,E2 -9399.352} C_VEL
LIN {X 0,Y 432.303,Z 271.448,A -85,B 0,C 180,E1 -9401.804,E2 -9401.804} C_VEL
LIN {X 0,Y 432.332,Z 271.445,A -85,B 0,C 180,E1 -9404.351,E2 -9404.351} C_VEL
LIN {X 0,Y 432.3,Z 271.448,A -85,B 0,C 180,E1 -9407.022,E2 -9407.022} C_VEL
LIN {X 0,Y 432.289,Z 271.449,A -85,B 0,C 180,E1 -9409.831,E2 -9409.831} C_VEL
LIN {X 0,Y 432.303,Z 271.447,A -85,B 0,C 180,E1 -9413.024,E2 -9413.024} C_VEL
LIN {X 0,Y 432.335,Z 271.443,A -85,B 0,C 180,E1 -9416.005,E2 -9416.005} C_VEL
LIN {X 0,Y 432.343,Z 271.443,A -85,B 0,C 180,E1 -9419.494,E2 -9419.494} C_VEL
LIN {X 0,Y 432.318,Z 271.445,A -85,B 0,C 180,E1 -9421.874,E2 -9421.874} C_VEL
LIN {X 0,Y 432.4,Z 271.554,A -85,B 0,C 180,E1 -9425.225,E2 -9425.225} C_VEL
LIN {X 0,Y 433.914,Z 280.914,A -85,B 0,C 180,E1 -9427.405,E2 -9427.405} C_VEL
LIN {X 0,Y 433.489,Z 291.988,A -85,B 0,C 180,E1 -9429.85,E2 -9429.85} C_VEL
LIN {X 0,Y 432.662,Z 308.373,A -85,B 0,C 180,E1 -9433.416,E2 -9433.416} C_VEL
LIN {X 0,Y 432.278,Z 319.244,A -85,B 0,C 180,E1 -9435.767,E2 -9435.767} C_VEL
LIN {X 0,Y 434.453,Z 339.494,A -85,B 0,C 180,E1 -9436.246,E2 -9436.246} C_VEL
LIN {X 0,Y 433.773,Z 398.167,A -85,B 0,C 180,E1 -9437.427,E2 -9437.427} C_VEL
LIN {X 0,Y 433.392,Z 410.999,A -85,B 0,C 180,E1 -9437.891,E2 -9437.891} C_VEL
LIN {X 0,Y 433.061,Z 420.771,A -85,B 0,C 180,E1 -9438.416,E2 -9438.416} C_VEL
LIN {X 0,Y 432.7,Z 429.224,A -85,B 0,C 180,E1 -9439,E2 -9439} C_VEL
LIN {X 0,Y 432.46,Z 437.424,A -85,B 0,C 180,E1 -9439.704,E2 -9439.704} C_VEL
LIN {X 0,Y 432.117,Z 445.232,A -85,B 0,C 180,E1 -9440.523,E2 -9440.523} C_VEL
LIN {X 0,Y 431.783,Z 453.431,A -85,B 0,C 180,E1 -9441.578,E2 -9441.578} C_VEL
LIN {X 0,Y 431.562,Z 460.563,A -85,B 0,C 180,E1 -9442.751,E2 -9442.751} C_VEL
LIN {X 0,Y 431.35,Z 466.325,A -85,B 0,C 180,E1 -9443.95,E2 -9443.95} C_VEL
LIN {X 0,Y 431.299,Z 471.461,A -85,B 0,C 180,E1 -9445.328,E2 -9445.328} C_VEL
LIN {X 0,Y 431.232,Z 475.249,A -85,B 0,C 180,E1 -9446.732,E2 -9446.732} C_VEL
LIN {X 0,Y 431.224,Z 477.603,A -85,B 0,C 180,E1 -9448.134,E2 -9448.134} C_VEL
LIN {X 0,Y 431.196,Z 478.546,A -85,B 0,C 180,E1 -9449.068,E2 -9449.068} C_VEL
LIN {X 0,Y 431.197,Z 478.87,A -85,B 0,C 180,E1 -9450.002,E2 -9450.002} C_VEL
LIN {X 0,Y 431.174,Z 478.654,A -85,B 0,C 180,E1 -9450.936,E2 -9450.936} C_VEL
LIN {X 0,Y 431.224,Z 477.936,A -85,B 0,C 180,E1 -9451.869,E2 -9451.869} C_VEL
LIN {X 0,Y 431.249,Z 476.703,A -85,B 0,C 180,E1 -9452.804,E2 -9452.804} C_VEL
LIN {X 0,Y 431.234,Z 473.716,A -85,B 0,C 180,E1 -9454.207,E2 -9454.207} C_VEL
LIN {X 0,Y 431.362,Z 469.423,A -85,B 0,C 180,E1 -9455.611,E2 -9455.611} C_VEL
LIN {X 0,Y 431.545,Z 463.602,A -85,B 0,C 180,E1 -9457.017,E2 -9457.017} C_VEL
LIN {X 0,Y 431.786,Z 457.233,A -85,B 0,C 180,E1 -9458.189,E2 -9458.189} C_VEL
LIN {X 0,Y 432.099,Z 451.028,A -85,B 0,C 180,E1 -9459.126,E2 -9459.126} C_VEL
LIN {X 0,Y 432.52,Z 443.497,A -85,B 0,C 180,E1 -9460.061,E2 -9460.061} C_VEL
LIN {X 0,Y 432.886,Z 435.461,A -85,B 0,C 180,E1 -9460.88,E2 -9460.88} C_VEL
LIN {X 0,Y 433.332,Z 425.516,A -85,B 0,C 180,E1 -9461.698,E2 -9461.698} C_VEL
LIN {X 0,Y 433.831,Z 414.015,A -85,B 0,C 180,E1 -9462.396,E2 -9462.396} C_VEL
LIN {X 0,Y 434.207,Z 404.98,A -85,B 0,C 180,E1 -9462.801,E2 -9462.801} C_VEL
LIN {X 0,Y 434.516,Z 395.197,A -85,B 0,C 180,E1 -9463.113,E2 -9463.113} C_VEL
LIN {X 0,Y 435.391,Z 337.715,A -85,B 0,C 180,E1 -9464.336,E2 -9464.336} C_VEL
LIN {X 0,Y 433.385,Z 322.206,A -85,B 0,C 180,E1 -9464.779,E2 -9464.779} C_VEL
LIN {X 0,Y 432.428,Z 316.494,A -85,B 0,C 180,E1 -9464.974,E2 -9464.974} C_VEL
LIN {X 0,Y 432.829,Z 300.808,A -85,B 0,C 180,E1 -9467.971,E2 -9467.971} C_VEL
LIN {X 0,Y 433.361,Z 284.009,A -85,B 0,C 180,E1 -9471.153,E2 -9471.153} C_VEL
LIN {X 0,Y 433.343,Z 276.456,A -85,B 0,C 180,E1 -9472.595,E2 -9472.595} C_VEL
LIN {X 0,Y 432.412,Z 271.437,A -85,B 0,C 180,E1 -9473.657,E2 -9473.657} C_VEL
LIN {X 0,Y 432.299,Z 271.455,A -85,B 0,C 180,E1 -9477.079,E2 -9477.079} C_VEL
LIN {X 0,Y 432.338,Z 271.446,A -85,B 0,C 180,E1 -9480.262,E2 -9480.262} C_VEL
LIN {X 0,Y 432.285,Z 271.45,A -85,B 0,C 180,E1 -9483.558,E2 -9483.558} C_VEL
LIN {X 0,Y 432.298,Z 271.451,A -85,B 0,C 180,E1 -9486.98,E2 -9486.98} C_VEL
LIN {X 0,Y 432.303,Z 271.444,A -85,B 0,C 180,E1 -9490.171,E2 -9490.171} C_VEL
LIN {X 0,Y 432.295,Z 271.45,A -85,B 0,C 180,E1 -9493.065,E2 -9493.065} C_VEL
LIN {X 0,Y 432.326,Z 271.441,A -85,B 0,C 180,E1 -9495.667,E2 -9495.667} C_VEL
LIN {X 0,Y 432.323,Z 271.441,A -85,B 0,C 180,E1 -9498.401,E2 -9498.401} C_VEL
LIN {X 0,Y 432.341,Z 271.438,A -85,B 0,C 180,E1 -9501.847,E2 -9501.847} C_VEL
LIN {X 0,Y 432.343,Z 271.442,A -85,B 0,C 180,E1 -9505.32,E2 -9505.32} C_VEL
LIN {X 0,Y 432.335,Z 271.445,A -85,B 0,C 180,E1 -9508.652,E2 -9508.652} C_VEL
LIN {X 0,Y 432.355,Z 271.441,A -85,B 0,C 180,E1 -9511.871,E2 -9511.871} C_VEL
LIN {X 0,Y 432.393,Z 271.442,A -85,B 0,C 180,E1 -9515.536,E2 -9515.536} C_VEL
LIN {X 0,Y 432.365,Z 271.445,A -85,B 0,C 180,E1 -9519.043,E2 -9519.043} C_VEL
LIN {X 0,Y 432.472,Z 271.43,A -85,B 0,C 180,E1 -9522.5,E2 -9522.5} C_VEL
LIN {X 0,Y 432.516,Z 271.604,A -85,B 0,C 180,E1 -9522.807,E2 -9522.807} C_VEL
LIN {X 0,Y 433.455,Z 275.59,A -85,B 0,C 180,E1 -9523.467,E2 -9523.467} C_VEL
LIN {X 0,Y 433.332,Z 286.642,A -85,B 0,C 180,E1 -9525.099,E2 -9525.099} C_VEL
LIN {X 0,Y 435.612,Z 300.299,A -85,B 0,C 180,E1 -9525.525,E2 -9525.525} C_VEL
LIN {X 0,Y 435.794,Z 306.342,A -85,B 0,C 180,E1 -9525.669,E2 -9525.669} C_VEL
LIN {X 0,Y 434.715,Z 366.965,A -85,B 0,C 180,E1 -9526.974,E2 -9526.974} C_VEL
LIN {X 0,Y 434.379,Z 378.489,A -85,B 0,C 180,E1 -9527.38,E2 -9527.38} C_VEL
LIN {X 0,Y 434.021,Z 389.322,A -85,B 0,C 180,E1 -9527.963,E2 -9527.963} C_VEL
LIN {X 0,Y 433.717,Z 397.705,A -85,B 0,C 180,E1 -9528.547,E2 -9528.547} C_VEL
LIN {X 0,Y 433.354,Z 405.861,A -85,B 0,C 180,E1 -9529.247,E2 -9529.247} C_VEL
LIN {X 0,Y 433.052,Z 413.628,A -85,B 0,C 180,E1 -9530.067,E2 -9530.067} C_VEL
LIN {X 0,Y 432.591,Z 421.779,A -85,B 0,C 180,E1 -9531.117,E2 -9531.117} C_VEL
LIN {X 0,Y 432.156,Z 428.895,A -85,B 0,C 180,E1 -9532.285,E2 -9532.285} C_VEL
LIN {X 0,Y 432.015,Z 434.498,A -85,B 0,C 180,E1 -9533.457,E2 -9533.457} C_VEL
LIN {X 0,Y 431.582,Z 439.716,A -85,B 0,C 180,E1 -9534.857,E2 -9534.857} C_VEL
LIN {X 0,Y 431.553,Z 443.496,A -85,B 0,C 180,E1 -9536.261,E2 -9536.261} C_VEL
LIN {X 0,Y 431.387,Z 445.2,A -85,B 0,C 180,E1 -9537.194,E2 -9537.194} C_VEL
LIN {X 0,Y 431.276,Z 446.374,A -85,B 0,C 180,E1 -9538.128,E2 -9538.128} C_VEL
LIN {X 0,Y 431.202,Z 447.043,A -85,B 0,C 180,E1 -9539.061,E2 -9539.061} C_VEL
LIN {X 0,Y 431.198,Z 447.214,A -85,B 0,C 180,E1 -9539.995,E2 -9539.995} C_VEL
LIN {X 0,Y 431.2,Z 446.828,A -85,B 0,C 180,E1 -9540.929,E2 -9540.929} C_VEL
LIN {X 0,Y 431.251,Z 445.842,A -85,B 0,C 180,E1 -9541.863,E2 -9541.863} C_VEL
LIN {X 0,Y 431.401,Z 443.458,A -85,B 0,C 180,E1 -9543.264,E2 -9543.264} C_VEL
LIN {X 0,Y 431.416,Z 439.664,A -85,B 0,C 180,E1 -9544.667,E2 -9544.667} C_VEL
LIN {X 0,Y 431.543,Z 436.388,A -85,B 0,C 180,E1 -9545.603,E2 -9545.603} C_VEL
LIN {X 0,Y 431.843,Z 430.501,A -85,B 0,C 180,E1 -9546.902,E2 -9546.902} C_VEL
LIN {X 0,Y 431.984,Z 424.625,A -85,B 0,C 180,E1 -9547.944,E2 -9547.944} C_VEL
LIN {X 0,Y 432.263,Z 418.187,A -85,B 0,C 180,E1 -9548.88,E2 -9548.88} C_VEL
LIN {X 0,Y 432.62,Z 409.321,A -85,B 0,C 180,E1 -9549.934,E2 -9549.934} C_VEL
LIN {X 0,Y 432.991,Z 399.063,A -85,B 0,C 180,E1 -9550.871,E2 -9550.871} C_VEL
LIN {X 0,Y 433.275,Z 391.005,A -85,B 0,C 180,E1 -9551.456,E2 -9551.456} C_VEL
LIN {X 0,Y 433.535,Z 381.806,A -85,B 0,C 180,E1 -9551.982,E2 -9551.982} C_VEL
LIN {X 0,Y 433.751,Z 372.252,A -85,B 0,C 180,E1 -9552.392,E2 -9552.392} C_VEL
LIN {X 0,Y 433.963,Z 362.269,A -85,B 0,C 180,E1 -9552.683,E2 -9552.683} C_VEL
LIN {X 0,Y 434.494,Z 301.984,A -85,B 0,C 180,E1 -9553.88,E2 -9553.88} C_VEL
LIN {X 0,Y 432.327,Z 288.21,A -85,B 0,C 180,E1 -9554.228,E2 -9554.228} C_VEL
LIN {X 0,Y 432.65,Z 277.758,A -85,B 0,C 180,E1 -9556.995,E2 -9556.995} C_VEL
LIN {X 0,Y 432.461,Z 271.43,A -85,B 0,C 180,E1 -9558.746,E2 -9558.746} C_VEL
LIN {X 0,Y 432.332,Z 271.443,A -85,B 0,C 180,E1 -9562.088,E2 -9562.088} C_VEL
LIN {X 0,Y 432.312,Z 271.447,A -85,B 0,C 180,E1 -9564.997,E2 -9564.997} C_VEL
LIN {X 0,Y 432.302,Z 271.447,A -85,B 0,C 180,E1 -9568.122,E2 -9568.122} C_VEL
LIN {X 0,Y 432.298,Z 271.448,A -85,B 0,C 180,E1 -9571.34,E2 -9571.34} C_VEL
LIN {X 0,Y 432.315,Z 271.446,A -85,B 0,C 180,E1 -9574.671,E2 -9574.671} C_VEL
LIN {X 0,Y 432.303,Z 271.448,A -85,B 0,C 180,E1 -9578.145,E2 -9578.145} C_VEL
LIN {X 0,Y 432.294,Z 271.449,A -85,B 0,C 180,E1 -9581.595,E2 -9581.595} C_VEL
LIN {X 0,Y 432.302,Z 271.448,A -85,B 0,C 180,E1 -9584.342,E2 -9584.342} C_VEL
LIN {X 0,Y 432.285,Z 271.45,A -85,B 0,C 180,E1 -9587.01,E2 -9587.01} C_VEL
LIN {X 0,Y 432.296,Z 271.448,A -85,B 0,C 180,E1 -9589.815,E2 -9589.815} C_VEL
LIN {X 0,Y 432.267,Z 271.452,A -85,B 0,C 180,E1 -9593.017,E2 -9593.017} C_VEL
LIN {X 0,Y 432.318,Z 271.446,A -85,B 0,C 180,E1 -9595.992,E2 -9595.992} C_VEL
LIN {X 0,Y 432.302,Z 271.448,A -85,B 0,C 180,E1 -9599.485,E2 -9599.485} C_VEL
LIN {X 0,Y 432.346,Z 271.442,A -85,B 0,C 180,E1 -9602.924,E2 -9602.924} C_VEL
LIN {X 0,Y 432.322,Z 271.446,A -85,B 0,C 180,E1 -9606.019,E2 -9606.019} C_VEL
LIN {X 0,Y 432.298,Z 271.448,A -85,B 0,C 180,E1 -9609.042,E2 -9609.042} C_VEL
LIN {X 0,Y 432.324,Z 271.447,A -85,B 0,C 180,E1 -9612.007,E2 -9612.007} C_VEL
LIN {X 0,Y 432.341,Z 271.444,A -85,B 0,C 180,E1 -9614.923,E2 -9614.923} C_VEL
LIN {X 0,Y 432.38,Z 271.436,A -85,B 0,C 180,E1 -9618.261,E2 -9618.261} C_VEL
LIN {X 0,Y 432.529,Z 271.421,A -85,B 0,C 180,E1 -9622.319,E2 -9622.319} C_VEL
LIN {X 0,Y 431.768,Z 271.515,A -85,B 0,C 180,E1 -9623.096,E2 -9623.096} C_VEL
LIN {X 0,Y 428.774,Z 271.889,A -85,B 0,C 180,E1 -9624.355,E2 -9624.355} C_VEL
LIN {X 0,Y 426.336,Z 272.193,A -85,B 0,C 180,E1 -9625.373,E2 -9625.373} C_VEL
LIN {X 0,Y 425.371,Z 272.312,A -85,B 0,C 180,E1 -9626.16,E2 -9626.16} C_VEL
LIN {X 0,Y 425.334,Z 272.315,A -85,B 0,C 180,E1 -9626.427,E2 -9626.427} C_VEL
LIN {X 0,Y 425.519,Z 272.293,A -85,B 0,C 180,E1 -9628.105,E2 -9628.105} C_VEL
LIN {X 0,Y 425.645,Z 272.277,A -85,B 0,C 180,E1 -9629.998,E2 -9629.998} C_VEL
LIN {X 0,Y 425.507,Z 272.294,A -85,B 0,C 180,E1 -9632.839,E2 -9632.839} C_VEL
LIN {X 0,Y 425.473,Z 272.301,A -85,B 0,C 180,E1 -9636.638,E2 -9636.638} C_VEL
LIN {X 0,Y 425.348,Z 272.314,A -85,B 0,C 180,E1 -9639.509,E2 -9639.509} C_VEL
LIN {X 0,Y 425.345,Z 272.316,A -85,B 0,C 180,E1 -9642.91,E2 -9642.91} C_VEL
LIN {X 0,Y 425.301,Z 272.32,A -85,B 0,C 180,E1 -9646.605,E2 -9646.605} C_VEL
LIN {X 0,Y 425.269,Z 272.323,A -85,B 0,C 180,E1 -9649.636,E2 -9649.636} C_VEL
LIN {X 0,Y 425.249,Z 272.327,A -85,B 0,C 180,E1 -9653.366,E2 -9653.366} C_VEL
LIN {X 0,Y 425.291,Z 272.321,A -85,B 0,C 180,E1 -9656.846,E2 -9656.846} C_VEL
LIN {X 0,Y 425.261,Z 272.324,A -85,B 0,C 180,E1 -9659.719,E2 -9659.719} C_VEL
LIN {X 0,Y 425.227,Z 272.329,A -85,B 0,C 180,E1 -9663.05,E2 -9663.05} C_VEL
LIN {X 0,Y 425.231,Z 272.328,A -85,B 0,C 180,E1 -9665.932,E2 -9665.932} C_VEL
LIN {X 0,Y 425.264,Z 272.324,A -85,B 0,C 180,E1 -9669.049,E2 -9669.049} C_VEL
LIN {X 0,Y 425.282,Z 272.323,A -85,B 0,C 180,E1 -9672.649,E2 -9672.649} C_VEL
LIN {X 0,Y 425.271,Z 272.324,A -85,B 0,C 180,E1 -9676.055,E2 -9676.055} C_VEL
LIN {X 0,Y 425.263,Z 272.325,A -85,B 0,C 180,E1 -9678.629,E2 -9678.629} C_VEL
LIN {X 0,Y 425.278,Z 272.322,A -85,B 0,C 180,E1 -9681.108,E2 -9681.108} C_VEL
LIN {X 0,Y 425.258,Z 272.325,A -85,B 0,C 180,E1 -9684.668,E2 -9684.668} C_VEL
LIN {X 0,Y 425.225,Z 272.331,A -85,B 0,C 180,E1 -9688.077,E2 -9688.077} C_VEL
LIN {X 0,Y 425.293,Z 272.321,A -85,B 0,C 180,E1 -9691.372,E2 -9691.372} C_VEL
LIN {X 0,Y 425.248,Z 272.326,A -85,B 0,C 180,E1 -9694.558,E2 -9694.558} C_VEL
LIN {X 0,Y 425.249,Z 272.326,A -85,B 0,C 180,E1 -9696.638,E2 -9696.638} C_VEL
LIN {X 0,Y 425.263,Z 272.324,A -85,B 0,C 180,E1 -9699.699,E2 -9699.699} C_VEL
LIN {X 0,Y 425.303,Z 272.32,A -85,B 0,C 180,E1 -9702.702,E2 -9702.702} C_VEL
LIN {X 0,Y 425.319,Z 272.318,A -85,B 0,C 180,E1 -9705.655,E2 -9705.655} C_VEL
LIN {X 0,Y 425.323,Z 272.319,A -85,B 0,C 180,E1 -9708.569,E2 -9708.569} C_VEL
LIN {X 0,Y 425.483,Z 272.297,A -85,B 0,C 180,E1 -9712.315,E2 -9712.315} C_VEL
LIN {X 0,Y 425.521,Z 272.292,A -85,B 0,C 180,E1 -9714.318,E2 -9714.318} C_VEL
LIN {X 0,Y 425.546,Z 272.289,A -85,B 0,C 180,E1 -9718.112,E2 -9718.112} C_VEL
LIN {X 0,Y 425.573,Z 272.286,A -85,B 0,C 180,E1 -9720.005,E2 -9720.005} C_VEL
LIN {X 0,Y 425.518,Z 272.294,A -85,B 0,C 180,E1 -9722.845,E2 -9722.845} C_VEL
LIN {X 0,Y 425.515,Z 272.293,A -85,B 0,C 180,E1 -9725.692,E2 -9725.692} C_VEL
LIN {X 0,Y 425.395,Z 272.308,A -85,B 0,C 180,E1 -9728.555,E2 -9728.555} C_VEL
LIN {X 0,Y 425.401,Z 272.307,A -85,B 0,C 180,E1 -9732.406,E2 -9732.406} C_VEL
LIN {X 0,Y 425.294,Z 272.323,A -85,B 0,C 180,E1 -9735.335,E2 -9735.335} C_VEL
LIN {X 0,Y 425.304,Z 272.32,A -85,B 0,C 180,E1 -9738.302,E2 -9738.302} C_VEL
LIN {X 0,Y 425.285,Z 272.323,A -85,B 0,C 180,E1 -9741.323,E2 -9741.323} C_VEL
LIN {X 0,Y 425.291,Z 272.321,A -85,B 0,C 180,E1 -9744.654,E2 -9744.654} C_VEL
LIN {X 0,Y 425.264,Z 272.326,A -85,B 0,C 180,E1 -9747.567,E2 -9747.567} C_VEL
LIN {X 0,Y 425.287,Z 272.322,A -85,B 0,C 180,E1 -9750.765,E2 -9750.765} C_VEL
LIN {X 0,Y 425.287,Z 272.321,A -85,B 0,C 180,E1 -9754.287,E2 -9754.287} C_VEL
LIN {X 0,Y 425.268,Z 272.324,A -85,B 0,C 180,E1 -9757.699,E2 -9757.699} C_VEL
LIN {X 0,Y 425.241,Z 272.327,A -85,B 0,C 180,E1 -9760.518,E2 -9760.518} C_VEL
LIN {X 0,Y 425.246,Z 272.326,A -85,B 0,C 180,E1 -9763.352,E2 -9763.352} C_VEL
LIN {X 0,Y 425.255,Z 272.327,A -85,B 0,C 180,E1 -9766.046,E2 -9766.046} C_VEL
LIN {X 0,Y 425.247,Z 272.326,A -85,B 0,C 180,E1 -9768.621,E2 -9768.621} C_VEL
LIN {X 0,Y 425.28,Z 272.322,A -85,B 0,C 180,E1 -9771.102,E2 -9771.102} C_VEL
LIN {X 0,Y 425.296,Z 272.321,A -85,B 0,C 180,E1 -9774.666,E2 -9774.666} C_VEL
LIN {X 0,Y 425.263,Z 272.324,A -85,B 0,C 180,E1 -9778.075,E2 -9778.075} C_VEL
LIN {X 0,Y 425.298,Z 272.32,A -85,B 0,C 180,E1 -9781.368,E2 -9781.368} C_VEL
LIN {X 0,Y 425.377,Z 272.39,A -85,B 0,C 180,E1 -9785.091,E2 -9785.091} C_VEL
LIN {X 0,Y 426.872,Z 281.394,A -85,B 0,C 180,E1 -9787.222,E2 -9787.222} C_VEL
LIN {X 0,Y 426.463,Z 292.656,A -85,B 0,C 180,E1 -9789.755,E2 -9789.755} C_VEL
LIN {X 0,Y 425.624,Z 308.575,A -85,B 0,C 180,E1 -9793.283,E2 -9793.283} C_VEL
LIN {X 0,Y 425.231,Z 319.063,A -85,B 0,C 180,E1 -9795.587,E2 -9795.587} C_VEL
LIN {X 0,Y 427.452,Z 340.519,A -85,B 0,C 180,E1 -9796.098,E2 -9796.098} C_VEL
LIN {X 0,Y 426.769,Z 397.719,A -85,B 0,C 180,E1 -9797.278,E2 -9797.278} C_VEL
LIN {X 0,Y 426.428,Z 409.431,A -85,B 0,C 180,E1 -9797.69,E2 -9797.69} C_VEL
LIN {X 0,Y 426.065,Z 419.486,A -85,B 0,C 180,E1 -9798.223,E2 -9798.223} C_VEL
LIN {X 0,Y 425.716,Z 428.139,A -85,B 0,C 180,E1 -9798.817,E2 -9798.817} C_VEL
LIN {X 0,Y 425.401,Z 436.478,A -85,B 0,C 180,E1 -9799.531,E2 -9799.531} C_VEL
LIN {X 0,Y 425.128,Z 444.414,A -85,B 0,C 180,E1 -9800.366,E2 -9800.366} C_VEL
LIN {X 0,Y 424.821,Z 450.974,A -85,B 0,C 180,E1 -9801.199,E2 -9801.199} C_VEL
LIN {X 0,Y 424.556,Z 458.684,A -85,B 0,C 180,E1 -9802.392,E2 -9802.392} C_VEL
LIN {X 0,Y 424.306,Z 464.938,A -85,B 0,C 180,E1 -9803.636,E2 -9803.636} C_VEL
LIN {X 0,Y 424.261,Z 469.439,A -85,B 0,C 180,E1 -9804.774,E2 -9804.774} C_VEL
LIN {X 0,Y 424.162,Z 472.481,A -85,B 0,C 180,E1 -9805.726,E2 -9805.726} C_VEL
LIN {X 0,Y 424.179,Z 475.751,A -85,B 0,C 180,E1 -9807.153,E2 -9807.153} C_VEL
LIN {X 0,Y 424.15,Z 477.276,A -85,B 0,C 180,E1 -9808.103,E2 -9808.103} C_VEL
LIN {X 0,Y 424.114,Z 478.234,A -85,B 0,C 180,E1 -9809.052,E2 -9809.052} C_VEL
LIN {X 0,Y 424.112,Z 478.578,A -85,B 0,C 180,E1 -9810.002,E2 -9810.002} C_VEL
LIN {X 0,Y 424.095,Z 478.4,A -85,B 0,C 180,E1 -9810.951,E2 -9810.951} C_VEL
LIN {X 0,Y 424.149,Z 477.719,A -85,B 0,C 180,E1 -9811.901,E2 -9811.901} C_VEL
LIN {X 0,Y 424.146,Z 476.522,A -85,B 0,C 180,E1 -9812.851,E2 -9812.851} C_VEL
LIN {X 0,Y 424.158,Z 473.574,A -85,B 0,C 180,E1 -9814.278,E2 -9814.278} C_VEL
LIN {X 0,Y 424.268,Z 469.305,A -85,B 0,C 180,E1 -9815.706,E2 -9815.706} C_VEL
LIN {X 0,Y 424.495,Z 463.54,A -85,B 0,C 180,E1 -9817.134,E2 -9817.134} C_VEL
LIN {X 0,Y 424.745,Z 457.221,A -85,B 0,C 180,E1 -9818.326,E2 -9818.326} C_VEL
LIN {X 0,Y 425.101,Z 451.053,A -85,B 0,C 180,E1 -9819.278,E2 -9819.278} C_VEL
LIN {X 0,Y 425.541,Z 443.562,A -85,B 0,C 180,E1 -9820.228,E2 -9820.228} C_VEL
LIN {X 0,Y 425.927,Z 435.641,A -85,B 0,C 180,E1 -9821.06,E2 -9821.06} C_VEL
LIN {X 0,Y 426.277,Z 428.855,A -85,B 0,C 180,E1 -9821.653,E2 -9821.653} C_VEL
LIN {X 0,Y 426.653,Z 420.657,A -85,B 0,C 180,E1 -9822.246,E2 -9822.246} C_VEL
LIN {X 0,Y 427.052,Z 411.321,A -85,B 0,C 180,E1 -9822.777,E2 -9822.777} C_VEL
LIN {X 0,Y 427.577,Z 400.056,A -85,B 0,C 180,E1 -9823.245,E2 -9823.245} C_VEL
LIN {X 0,Y 427.96,Z 383.343,A -85,B 0,C 180,E1 -9823.648,E2 -9823.648} C_VEL
LIN {X 0,Y 428.672,Z 338.345,A -85,B 0,C 180,E1 -9824.624,E2 -9824.624} C_VEL
LIN {X 0,Y 426.731,Z 323.402,A -85,B 0,C 180,E1 -9825.07,E2 -9825.07} C_VEL
LIN {X 0,Y 425.508,Z 316.135,A -85,B 0,C 180,E1 -9825.325,E2 -9825.325} C_VEL
LIN {X 0,Y 426.034,Z 298.324,A -85,B 0,C 180,E1 -9828.766,E2 -9828.766} C_VEL
LIN {X 0,Y 426.498,Z 282.797,A -85,B 0,C 180,E1 -9831.764,E2 -9831.764} C_VEL
LIN {X 0,Y 426.301,Z 277.01,A -85,B 0,C 180,E1 -9832.902,E2 -9832.902} C_VEL
LIN {X 0,Y 425.334,Z 272.319,A -85,B 0,C 180,E1 -9833.882,E2 -9833.882} C_VEL
LIN {X 0,Y 425.249,Z 272.331,A -85,B 0,C 180,E1 -9837.566,E2 -9837.566} C_VEL
LIN {X 0,Y 425.283,Z 272.324,A -85,B 0,C 180,E1 -9839.721,E2 -9839.721} C_VEL
LIN {X 0,Y 425.243,Z 272.329,A -85,B 0,C 180,E1 -9843.053,E2 -9843.053} C_VEL
LIN {X 0,Y 425.247,Z 272.327,A -85,B 0,C 180,E1 -9846.512,E2 -9846.512} C_VEL
LIN {X 0,Y 425.258,Z 272.328,A -85,B 0,C 180,E1 -9849.033,E2 -9849.033} C_VEL
LIN {X 0,Y 425.258,Z 272.322,A -85,B 0,C 180,E1 -9851.95,E2 -9851.95} C_VEL
LIN {X 0,Y 425.281,Z 272.321,A -85,B 0,C 180,E1 -9855.285,E2 -9855.285} C_VEL
LIN {X 0,Y 425.263,Z 272.322,A -85,B 0,C 180,E1 -9858.617,E2 -9858.617} C_VEL
LIN {X 0,Y 425.294,Z 272.32,A -85,B 0,C 180,E1 -9861.097,E2 -9861.097} C_VEL
LIN {X 0,Y 425.31,Z 272.317,A -85,B 0,C 180,E1 -9864.662,E2 -9864.662} C_VEL
LIN {X 0,Y 425.279,Z 272.321,A -85,B 0,C 180,E1 -9868.071,E2 -9868.071} C_VEL
LIN {X 0,Y 425.322,Z 272.321,A -85,B 0,C 180,E1 -9871.364,E2 -9871.364} C_VEL
LIN {X 0,Y 425.285,Z 272.326,A -85,B 0,C 180,E1 -9874.55,E2 -9874.55} C_VEL
LIN {X 0,Y 425.299,Z 272.324,A -85,B 0,C 180,E1 -9876.631,E2 -9876.631} C_VEL
LIN {X 0,Y 425.31,Z 272.321,A -85,B 0,C 180,E1 -9879.691,E2 -9879.691} C_VEL
LIN {X 0,Y 425.468,Z 272.448,A -85,B 0,C 180,E1 -9882.482,E2 -9882.482} C_VEL
LIN {X 0,Y 426.737,Z 278.589,A -85,B 0,C 180,E1 -9883.514,E2 -9883.514} C_VEL
LIN {X 0,Y 426.503,Z 286.599,A -85,B 0,C 180,E1 -9884.736,E2 -9884.736} C_VEL
LIN {X 0,Y 429.006,Z 301.549,A -85,B 0,C 180,E1 -9885.231,E2 -9885.231} C_VEL
LIN {X 0,Y 428.85,Z 320.625,A -85,B 0,C 180,E1 -9885.675,E2 -9885.675} C_VEL
LIN {X 0,Y 427.921,Z 367.339,A -85,B 0,C 180,E1 -9886.703,E2 -9886.703} C_VEL
LIN {X 0,Y 427.586,Z 378.814,A -85,B 0,C 180,E1 -9887.115,E2 -9887.115} C_VEL
LIN {X 0,Y 427.211,Z 388.735,A -85,B 0,C 180,E1 -9887.647,E2 -9887.647} C_VEL
LIN {X 0,Y 426.951,Z 397.266,A -85,B 0,C 180,E1 -9888.242,E2 -9888.242} C_VEL
LIN {X 0,Y 426.451,Z 405.527,A -85,B 0,C 180,E1 -9888.951,E2 -9888.951} C_VEL
LIN {X 0,Y 426.173,Z 413.357,A -85,B 0,C 180,E1 -9889.785,E2 -9889.785} C_VEL
LIN {X 0,Y 425.72,Z 420.714,A -85,B 0,C 180,E1 -9890.733,E2 -9890.733} C_VEL
LIN {X 0,Y 425.248,Z 428.18,A -85,B 0,C 180,E1 -9891.92,E2 -9891.92} C_VEL
LIN {X 0,Y 424.987,Z 434.99,A -85,B 0,C 180,E1 -9893.348,E2 -9893.348} C_VEL
LIN {X 0,Y 424.598,Z 438.633,A -85,B 0,C 180,E1 -9894.296,E2 -9894.296} C_VEL
LIN {X 0,Y 424.548,Z 442.754,A -85,B 0,C 180,E1 -9895.723,E2 -9895.723} C_VEL
LIN {X 0,Y 424.501,Z 443.906,A -85,B 0,C 180,E1 -9896.198,E2 -9896.198} C_VEL
LIN {X 0,Y 424.324,Z 445.586,A -85,B 0,C 180,E1 -9897.147,E2 -9897.147} C_VEL
LIN {X 0,Y 424.201,Z 446.719,A -85,B 0,C 180,E1 -9898.096,E2 -9898.096} C_VEL
LIN {X 0,Y 424.121,Z 447.344,A -85,B 0,C 180,E1 -9899.046,E2 -9899.046} C_VEL
LIN {X 0,Y 424.114,Z 447.467,A -85,B 0,C 180,E1 -9899.995,E2 -9899.995} C_VEL
LIN {X 0,Y 424.118,Z 447.059,A -85,B 0,C 180,E1 -9900.945,E2 -9900.945} C_VEL
LIN {X 0,Y 424.178,Z 446.04,A -85,B 0,C 180,E1 -9901.894,E2 -9901.894} C_VEL
LIN {X 0,Y 424.334,Z 443.576,A -85,B 0,C 180,E1 -9903.318,E2 -9903.318} C_VEL
LIN {X 0,Y 424.344,Z 439.693,A -85,B 0,C 180,E1 -9904.745,E2 -9904.745} C_VEL
LIN {X 0,Y 424.583,Z 434.367,A -85,B 0,C 180,E1 -9906.171,E2 -9906.171} C_VEL
LIN {X 0,Y 424.825,Z 428.641,A -85,B 0,C 180,E1 -9907.361,E2 -9907.361} C_VEL
LIN {X 0,Y 425.064,Z 421.394,A -85,B 0,C 180,E1 -9908.552,E2 -9908.552} C_VEL
LIN {X 0,Y 425.405,Z 413.095,A -85,B 0,C 180,E1 -9909.624,E2 -9909.624} C_VEL
LIN {X 0,Y 425.758,Z 405.184,A -85,B 0,C 180,E1 -9910.456,E2 -9910.456} C_VEL
LIN {X 0,Y 426.004,Z 396.863,A -85,B 0,C 180,E1 -9911.172,E2 -9911.172} C_VEL
